KUKA KRL program: f1_Kuka_APT230T02S30.SRC

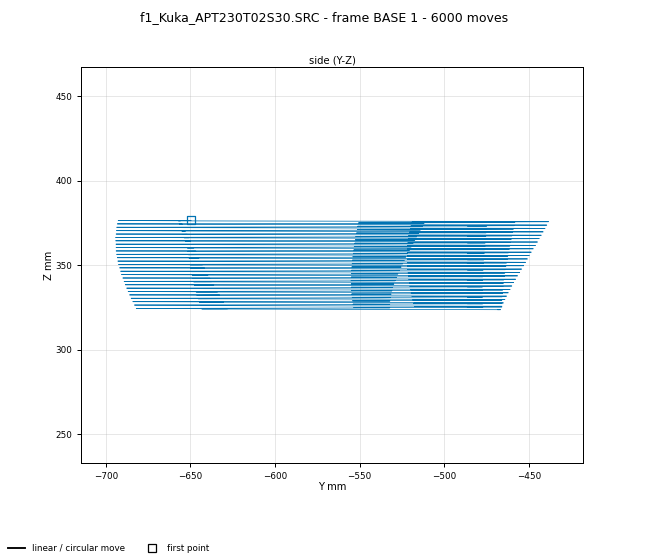
[picture p0: tool path of f1_Kuka_APT230T02S30.SRC in frame BASE 1, 6000 of 6001 moves have a stored position in this frame; points joined in program order, loops and branches not executed]
&ACCESS RVP
&REL 2
&PARAM TEMPLATE = C:\KRC\Roboter\Template\vorgabe
&PARAM EDITMASK = *
DEF f1_Kuka_APT230T02S30()


;FOLD INI;%{PE}%V3.2.0,%MKUKATPBASIS,%CINIT,%VCOMMON,%P
  ;FOLD BAS INI;%{E}%V3.2.0,%MKUKATPBASIS,%CINIT,%VINIT,%P
    GLOBAL INTERRUPT DECL 3 WHEN $STOPMESS==TRUE DO IR_STOPM ( )
    INTERRUPT ON 3
    BAS (#INITMOV,0 )
  ;ENDFOLD (BAS INI)
  ;FOLD USER INI;%{E}%V3.2.0,%MKUKATPUSER,%CINIT,%VINIT,%P
    ;Make your modifications here
  ;ENDFOLD (USER INI)
;ENDFOLD (INI)


;*** Make Null PTP Move
  PTP $pos_act

;*** Auto Load The Correct TOOL Data
  $tool=tool_data[2]

;*** Auto Load The Correct BASE Data
  $base=base_data[1]

  $ADVANCE = 5

;*** Restate Last Velocity
MMPM(30000.0)
SetRPM(8000)
LIN {X 0.163,Y -649.704,Z 376.543,A 0.000,B 0.000,C 90.000,E1 313.704} C_DIS
LIN {X -0.056,Y -653.378,Z 376.537,A 0.000,B 0.000,C 90.000,E1 312.732} C_DIS
LIN {X 0.228,Y -658.806,Z 376.529,A 0.000,B 0.000,C 90.000,E1 311.229} C_DIS
LIN {X 0.152,Y -663.209,Z 376.522,A 0.000,B 0.000,C 90.000,E1 310.011} C_DIS
LIN {X 0.173,Y -665.779,Z 376.518,A 0.000,B 0.000,C 90.000,E1 309.277} C_DIS
LIN {X -0.223,Y -669.831,Z 376.512,A 0.000,B 0.000,C 90.000,E1 308.096} C_DIS
LIN {X -0.019,Y -673.030,Z 376.506,A 0.000,B 0.000,C 90.000,E1 307.111} C_DIS
LIN {X 0.091,Y -676.010,Z 376.501,A 0.000,B 0.000,C 90.000,E1 306.137} C_DIS
LIN {X -0.172,Y -678.143,Z 376.497,A 0.000,B 0.000,C 90.000,E1 305.438} C_DIS
LIN {X 0.146,Y -680.171,Z 376.493,A 0.000,B 0.000,C 90.000,E1 304.692} C_DIS
LIN {X 0.314,Y -681.620,Z 376.490,A 0.000,B 0.000,C 90.000,E1 304.199} C_DIS
LIN {X -0.083,Y -684.557,Z 376.484,A 0.000,B 0.000,C 90.000,E1 303.038} C_DIS
LIN {X 0.141,Y -687.938,Z 376.476,A 0.000,B 0.000,C 90.000,E1 301.592} C_DIS
LIN {X 0.208,Y -689.459,Z 376.472,A 0.000,B 0.000,C 90.000,E1 300.875} C_DIS
LIN {X -0.299,Y -690.732,Z 376.468,A 0.000,B 0.000,C 90.000,E1 300.207} C_DIS
LIN {X 0.146,Y -691.673,Z 376.464,A 0.000,B 0.000,C 90.000,E1 299.461} C_DIS
LIN {X 0.255,Y -692.307,Z 376.460,A 0.000,B 0.000,C 90.000,E1 298.743} C_DIS
LIN {X 0.046,Y -692.607,Z 376.456,A 0.000,B 0.000,C 90.000,E1 298.052} C_DIS
LIN {X -0.076,Y -692.747,Z 376.453,A 0.000,B 0.000,C 90.000,E1 297.590} C_DIS
LIN {X 0.045,Y -692.691,Z 376.449,A 0.000,B 0.000,C 90.000,E1 296.873} C_DIS
LIN {X 0.291,Y -692.484,Z 376.448,A 0.000,B 0.000,C 90.000,E1 296.616} C_DIS
LIN {X 0.159,Y -692.369,Z 376.445,A 0.000,B 0.000,C 90.000,E1 296.155} C_DIS
LIN {X 0.154,Y -691.580,Z 376.439,A 0.000,B 0.000,C 90.000,E1 294.975} C_DIS
LIN {X 0.199,Y -690.341,Z 376.434,A 0.000,B 0.000,C 90.000,E1 294.027} C_DIS
LIN {X 0.179,Y -688.376,Z 376.427,A 0.000,B 0.000,C 90.000,E1 292.845} C_DIS
LIN {X 0.168,Y -686.612,Z 376.422,A 0.000,B 0.000,C 90.000,E1 291.897} C_DIS
LIN {X 0.028,Y -683.516,Z 376.414,A 0.000,B 0.000,C 90.000,E1 290.482} C_DIS
LIN {X 0.281,Y -680.993,Z 376.407,A 0.000,B 0.000,C 90.000,E1 289.268} C_DIS
LIN {X -0.153,Y -678.267,Z 376.401,A 0.000,B 0.000,C 90.000,E1 288.109} C_DIS
LIN {X -0.199,Y -675.630,Z 376.394,A 0.000,B 0.000,C 90.000,E1 286.913} C_DIS
LIN {X 0.305,Y -672.527,Z 376.386,A 0.000,B 0.000,C 90.000,E1 285.426} C_DIS
LIN {X 0.074,Y -666.335,Z 376.368,A 0.000,B 0.000,C 90.000,E1 282.299} C_DIS
LIN {X -0.156,Y -661.494,Z 376.351,A 0.000,B 0.000,C 90.000,E1 279.151} C_DIS
LIN {X 0.314,Y -657.922,Z 376.332,A 0.000,B 0.000,C 90.000,E1 275.682} C_DIS
LIN {X -0.180,Y -656.502,Z 376.318,A 0.000,B 0.000,C 90.000,E1 273.269} C_DIS
LIN {X -0.289,Y -655.863,Z 376.303,A 0.000,B 0.000,C 90.000,E1 270.573} C_DIS
LIN {X -0.067,Y -655.914,Z 376.291,A 0.000,B 0.000,C 90.000,E1 268.339} C_DIS
LIN {X 0.196,Y -656.501,Z 376.279,A 0.000,B 0.000,C 90.000,E1 266.102} C_DIS
LIN {X 0.156,Y -656.858,Z 376.273,A 0.000,B 0.000,C 90.000,E1 265.122} C_DIS
LIN {X 0.066,Y -657.098,Z 376.268,A 0.000,B 0.000,C 90.000,E1 264.147} C_DIS
LIN {X -0.089,Y -657.122,Z 376.261,A 0.000,B 0.000,C 90.000,E1 262.932} C_DIS
LIN {X 0.014,Y -656.948,Z 376.257,A 0.000,B 0.000,C 90.000,E1 262.186} C_DIS
LIN {X 0.078,Y -656.478,Z 376.251,A 0.000,B 0.000,C 90.000,E1 261.197} C_DIS
LIN {X -0.265,Y -656.044,Z 376.248,A 0.000,B 0.000,C 90.000,E1 260.735} C_DIS
LIN {X -0.049,Y -653.895,Z 376.239,A 0.000,B 0.000,C 90.000,E1 258.993} C_DIS
LIN {X -0.171,Y -653.502,Z 376.238,A 0.000,B 0.000,C 90.000,E1 258.757} C_DIS
LIN {X 0.226,Y -653.064,Z 376.235,A 0.000,B 0.000,C 90.000,E1 258.229} C_DIS
LIN {X -0.141,Y -651.961,Z 376.231,A 0.000,B 0.000,C 90.000,E1 257.521} C_DIS
LIN {X 0.248,Y -651.310,Z 376.228,A 0.000,B 0.000,C 90.000,E1 256.992} C_DIS
LIN {X 0.374,Y -649.587,Z 376.222,A 0.000,B 0.000,C 90.000,E1 255.992} C_DIS
LIN {X 0.113,Y -648.593,Z 376.220,A 0.000,B 0.000,C 90.000,E1 255.519} C_DIS
LIN {X 0.195,Y -646.368,Z 376.214,A 0.000,B 0.000,C 90.000,E1 254.519} C_DIS
LIN {X -0.057,Y -644.432,Z 376.210,A 0.000,B 0.000,C 90.000,E1 253.795} C_DIS
LIN {X 0.107,Y -642.226,Z 376.206,A 0.000,B 0.000,C 90.000,E1 253.032} C_DIS
LIN {X -0.149,Y -639.008,Z 376.200,A 0.000,B 0.000,C 90.000,E1 252.054} C_DIS
LIN {X 0.143,Y -636.488,Z 376.196,A 0.000,B 0.000,C 90.000,E1 251.275} C_DIS
LIN {X -0.170,Y -632.779,Z 376.190,A 0.000,B 0.000,C 90.000,E1 250.296} C_DIS
LIN {X -0.147,Y -627.965,Z 376.183,A 0.000,B 0.000,C 90.000,E1 249.028} C_DIS
LIN {X 0.239,Y -623.929,Z 376.178,A 0.000,B 0.000,C 90.000,E1 247.975} C_DIS
LIN {X -0.254,Y -618.652,Z 376.171,A 0.000,B 0.000,C 90.000,E1 246.741} C_DIS
LIN {X 0.226,Y -613.303,Z 376.164,A 0.000,B 0.000,C 90.000,E1 245.409} C_DIS
LIN {X -0.239,Y -606.742,Z 376.155,A 0.000,B 0.000,C 90.000,E1 243.896} C_DIS
LIN {X 0.242,Y -600.208,Z 376.146,A 0.000,B 0.000,C 90.000,E1 242.281} C_DIS
LIN {X -0.034,Y -592.621,Z 376.136,A 0.000,B 0.000,C 90.000,E1 240.461} C_DIS
LIN {X -0.159,Y -583.246,Z 376.123,A 0.000,B 0.000,C 90.000,E1 238.074} C_DIS
LIN {X 0.202,Y -575.502,Z 376.111,A 0.000,B 0.000,C 90.000,E1 235.881} C_DIS
LIN {X -0.064,Y -569.970,Z 376.102,A 0.000,B 0.000,C 90.000,E1 234.276} C_DIS
LIN {X -0.226,Y -565.448,Z 376.094,A 0.000,B 0.000,C 90.000,E1 232.924} C_DIS
LIN {X -0.227,Y -561.722,Z 376.088,A 0.000,B 0.000,C 90.000,E1 231.823} C_DIS
LIN {X -0.109,Y -555.912,Z 376.079,A 0.000,B 0.000,C 90.000,E1 230.150} C_DIS
LIN {X 0.223,Y -549.385,Z 376.068,A 0.000,B 0.000,C 90.000,E1 228.162} C_DIS
LIN {X -0.030,Y -544.865,Z 376.060,A 0.000,B 0.000,C 90.000,E1 226.782} C_DIS
LIN {X 0.002,Y -540.354,Z 376.052,A 0.000,B 0.000,C 90.000,E1 225.364} C_DIS
LIN {X -0.058,Y -534.992,Z 376.043,A 0.000,B 0.000,C 90.000,E1 223.662} C_DIS
LIN {X 0.145,Y -529.675,Z 376.033,A 0.000,B 0.000,C 90.000,E1 221.919} C_DIS
LIN {X -0.215,Y -522.839,Z 376.020,A 0.000,B 0.000,C 90.000,E1 219.644} C_DIS
LIN {X -0.174,Y -517.905,Z 376.010,A 0.000,B 0.000,C 90.000,E1 217.890} C_DIS
LIN {X 0.166,Y -513.141,Z 376.001,A 0.000,B 0.000,C 90.000,E1 216.091} C_DIS
LIN {X -0.003,Y -507.832,Z 375.989,A 0.000,B 0.000,C 90.000,E1 214.040} C_DIS
LIN {X -0.025,Y -502.737,Z 375.978,A 0.000,B 0.000,C 90.000,E1 211.957} C_DIS
LIN {X 0.071,Y -499.981,Z 375.971,A 0.000,B 0.000,C 90.000,E1 210.747} C_DIS
LIN {X 0.005,Y -495.857,Z 375.961,A 0.000,B 0.000,C 90.000,E1 208.949} C_DIS
LIN {X 0.061,Y -491.070,Z 375.949,A 0.000,B 0.000,C 90.000,E1 206.821} C_DIS
LIN {X -0.019,Y -486.141,Z 375.937,A 0.000,B 0.000,C 90.000,E1 204.695} C_DIS
LIN {X 0.039,Y -482.460,Z 375.929,A 0.000,B 0.000,C 90.000,E1 203.153} C_DIS
LIN {X 0.222,Y -478.781,Z 375.920,A 0.000,B 0.000,C 90.000,E1 201.589} C_DIS
LIN {X -0.045,Y -474.447,Z 375.910,A 0.000,B 0.000,C 90.000,E1 199.758} C_DIS
LIN {X -0.204,Y -468.870,Z 375.896,A 0.000,B 0.000,C 90.000,E1 197.275} C_DIS
LIN {X -0.082,Y -464.978,Z 375.885,A 0.000,B 0.000,C 90.000,E1 195.371} C_DIS
LIN {X 0.184,Y -460.689,Z 375.873,A 0.000,B 0.000,C 90.000,E1 193.119} C_DIS
LIN {X 0.121,Y -455.523,Z 375.857,A 0.000,B 0.000,C 90.000,E1 190.254} C_DIS
LIN {X -0.237,Y -451.787,Z 375.845,A 0.000,B 0.000,C 90.000,E1 188.049} C_DIS
LIN {X 0.137,Y -448.336,Z 375.832,A 0.000,B 0.000,C 90.000,E1 185.739} C_DIS
LIN {X -0.039,Y -442.797,Z 375.807,A 0.000,B 0.000,C 90.000,E1 181.203} C_DIS
LIN {X -0.001,Y -439.945,Z 375.787,A 0.000,B 0.000,C 90.000,E1 177.593} C_DIS
LIN {X -0.171,Y -438.299,Z 375.763,A 0.000,B 0.000,C 90.000,E1 173.337} C_DIS
LIN {X -0.004,Y -438.509,Z 375.737,A 0.000,B 0.000,C 90.000,E1 168.701} C_DIS
LIN {X 0.032,Y -442.330,Z 375.704,A 0.000,B 0.000,C 90.000,E1 162.779} C_DIS
LIN {X -0.158,Y -446.351,Z 375.684,A 0.000,B 0.000,C 90.000,E1 159.209} C_DIS
LIN {X 0.123,Y -452.263,Z 375.663,A 0.000,B 0.000,C 90.000,E1 155.281} C_DIS
LIN {X -0.157,Y -455.693,Z 375.652,A 0.000,B 0.000,C 90.000,E1 153.384} C_DIS
LIN {X -0.048,Y -463.942,Z 375.631,A 0.000,B 0.000,C 90.000,E1 149.537} C_DIS
LIN {X -0.201,Y -473.215,Z 375.612,A 0.000,B 0.000,C 90.000,E1 146.087} C_DIS
LIN {X -0.040,Y -481.024,Z 375.598,A 0.000,B 0.000,C 90.000,E1 143.577} C_DIS
LIN {X -0.174,Y -487.223,Z 375.587,A 0.000,B 0.000,C 90.000,E1 141.743} C_DIS
LIN {X -0.003,Y -492.431,Z 375.579,A 0.000,B 0.000,C 90.000,E1 140.194} C_DIS
LIN {X 0.032,Y -496.524,Z 375.572,A 0.000,B 0.000,C 90.000,E1 138.976} C_DIS
LIN {X 0.131,Y -500.477,Z 375.565,A 0.000,B 0.000,C 90.000,E1 137.757} C_DIS
LIN {X -0.085,Y -504.202,Z 375.559,A 0.000,B 0.000,C 90.000,E1 136.581} C_DIS
LIN {X 0.236,Y -506.818,Z 375.554,A 0.000,B 0.000,C 90.000,E1 135.648} C_DIS
LIN {X -0.258,Y -509.980,Z 375.547,A 0.000,B 0.000,C 90.000,E1 134.514} C_DIS
LIN {X 0.233,Y -511.429,Z 375.544,A 0.000,B 0.000,C 90.000,E1 133.866} C_DIS
LIN {X -0.086,Y -513.399,Z 375.539,A 0.000,B 0.000,C 90.000,E1 133.014} C_DIS
LIN {X 0.085,Y -514.607,Z 375.536,A 0.000,B 0.000,C 90.000,E1 132.405} C_DIS
LIN {X 0.145,Y -516.140,Z 375.531,A 0.000,B 0.000,C 90.000,E1 131.515} C_DIS
LIN {X 0.265,Y -517.444,Z 375.526,A 0.000,B 0.000,C 90.000,E1 130.620} C_DIS
LIN {X 0.003,Y -518.419,Z 375.521,A 0.000,B 0.000,C 90.000,E1 129.769} C_DIS
LIN {X 0.085,Y -519.013,Z 375.514,A 0.000,B 0.000,C 90.000,E1 128.588} C_DIS
LIN {X -0.144,Y -518.670,Z 375.508,A 0.000,B 0.000,C 90.000,E1 127.443} C_DIS
LIN {X -0.317,Y -518.081,Z 375.503,A 0.000,B 0.000,C 90.000,E1 126.583} C_DIS
LIN {X -0.016,Y -517.558,Z 375.500,A 0.000,B 0.000,C 90.000,E1 125.964} C_DIS
LIN {X -0.199,Y -516.417,Z 375.495,A 0.000,B 0.000,C 90.000,E1 125.105} C_DIS
LIN {X 0.025,Y -515.035,Z 375.490,A 0.000,B 0.000,C 90.000,E1 124.199} C_DIS
LIN {X 0.230,Y -513.407,Z 375.485,A 0.000,B 0.000,C 90.000,E1 123.293} C_DIS
LIN {X 0.135,Y -511.551,Z 375.480,A 0.000,B 0.000,C 90.000,E1 122.418} C_DIS
LIN {X 0.025,Y -509.351,Z 375.475,A 0.000,B 0.000,C 90.000,E1 121.544} C_DIS
LIN {X 0.215,Y -505.989,Z 375.469,A 0.000,B 0.000,C 90.000,E1 120.335} C_DIS
LIN {X 0.037,Y -503.218,Z 375.464,A 0.000,B 0.000,C 90.000,E1 119.461} C_DIS
LIN {X -0.036,Y -501.245,Z 375.460,A 0.000,B 0.000,C 90.000,E1 118.871} C_DIS
LIN {X -0.070,Y -497.929,Z 375.455,A 0.000,B 0.000,C 90.000,E1 117.975} C_DIS
LIN {X 0.091,Y -494.389,Z 375.450,A 0.000,B 0.000,C 90.000,E1 117.052} C_DIS
LIN {X 0.008,Y -489.325,Z 375.444,A 0.000,B 0.000,C 90.000,E1 115.848} C_DIS
LIN {X -0.162,Y -485.364,Z 375.439,A 0.000,B 0.000,C 90.000,E1 114.951} C_DIS
LIN {X -0.137,Y -481.107,Z 375.433,A 0.000,B 0.000,C 90.000,E1 114.027} C_DIS
LIN {X 0.019,Y -475.347,Z 375.427,A 0.000,B 0.000,C 90.000,E1 112.770} C_DIS
LIN {X 0.096,Y -468.465,Z 375.419,A 0.000,B 0.000,C 90.000,E1 111.354} C_DIS
LIN {X 0.172,Y -458.226,Z 375.407,A 0.000,B 0.000,C 90.000,E1 109.268} C_DIS
LIN {X 0.132,Y -458.213,Z 375.407,A 0.000,B 0.000,C 90.000,E1 109.268} C_DIS
LIN {X -0.112,Y -467.081,Z 375.384,A 0.000,B 0.000,C 90.000,E1 105.190} C_DIS
LIN {X 0.263,Y -467.845,Z 375.383,A 0.000,B 0.000,C 90.000,E1 104.828} C_DIS
LIN {X -0.176,Y -475.403,Z 375.358,A 0.000,B 0.000,C 90.000,E1 100.489} C_DIS
LIN {X 0.130,Y -476.055,Z 375.356,A 0.000,B 0.000,C 90.000,E1 100.141} C_DIS
LIN {X -0.066,Y -481.981,Z 375.331,A 0.000,B 0.000,C 90.000,E1 95.511} C_DIS
LIN {X 0.068,Y -482.357,Z 375.327,A 0.000,B 0.000,C 90.000,E1 94.878} C_DIS
LIN {X 0.205,Y -485.435,Z 375.305,A 0.000,B 0.000,C 90.000,E1 90.859} C_DIS
LIN {X -0.143,Y -485.505,Z 375.302,A 0.000,B 0.000,C 90.000,E1 90.286} C_DIS
LIN {X 0.238,Y -486.377,Z 375.281,A 0.000,B 0.000,C 90.000,E1 86.560} C_DIS
LIN {X 0.062,Y -486.365,Z 375.279,A 0.000,B 0.000,C 90.000,E1 86.274} C_DIS
LIN {X 0.151,Y -484.691,Z 375.254,A 0.000,B 0.000,C 90.000,E1 81.659} C_DIS
LIN {X -0.052,Y -484.454,Z 375.252,A 0.000,B 0.000,C 90.000,E1 81.376} C_DIS
LIN {X -0.048,Y -480.646,Z 375.228,A 0.000,B 0.000,C 90.000,E1 77.061} C_DIS
LIN {X -0.081,Y -480.368,Z 375.226,A 0.000,B 0.000,C 90.000,E1 76.756} C_DIS
LIN {X 0.233,Y -474.654,Z 375.203,A 0.000,B 0.000,C 90.000,E1 72.543} C_DIS
LIN {X 0.192,Y -474.657,Z 375.203,A 0.000,B 0.000,C 90.000,E1 72.543} C_DIS
LIN {X -0.287,Y -485.495,Z 375.195,A 0.000,B 0.000,C 90.000,E1 71.040} C_DIS
LIN {X 0.252,Y -493.631,Z 375.188,A 0.000,B 0.000,C 90.000,E1 69.752} C_DIS
LIN {X -0.242,Y -499.267,Z 375.183,A 0.000,B 0.000,C 90.000,E1 68.901} C_DIS
LIN {X 0.087,Y -501.950,Z 375.180,A 0.000,B 0.000,C 90.000,E1 68.411} C_DIS
LIN {X 0.051,Y -506.035,Z 375.176,A 0.000,B 0.000,C 90.000,E1 67.667} C_DIS
LIN {X 0.236,Y -509.004,Z 375.173,A 0.000,B 0.000,C 90.000,E1 67.050} C_DIS
LIN {X 0.155,Y -511.255,Z 375.170,A 0.000,B 0.000,C 90.000,E1 66.613} C_DIS
LIN {X 0.087,Y -513.235,Z 375.168,A 0.000,B 0.000,C 90.000,E1 66.177} C_DIS
LIN {X -0.091,Y -514.004,Z 375.167,A 0.000,B 0.000,C 90.000,E1 66.049} C_DIS
LIN {X -0.146,Y -515.847,Z 375.164,A 0.000,B 0.000,C 90.000,E1 65.613} C_DIS
LIN {X -0.322,Y -516.567,Z 375.164,A 0.000,B 0.000,C 90.000,E1 65.485} C_DIS
LIN {X -0.179,Y -519.975,Z 375.159,A 0.000,B 0.000,C 90.000,E1 64.588} C_DIS
LIN {X 0.099,Y -522.152,Z 375.156,A 0.000,B 0.000,C 90.000,E1 63.973} C_DIS
LIN {X 0.153,Y -524.176,Z 375.152,A 0.000,B 0.000,C 90.000,E1 63.384} C_DIS
LIN {X -0.085,Y -526.875,Z 375.147,A 0.000,B 0.000,C 90.000,E1 62.538} C_DIS
LIN {X -0.128,Y -530.387,Z 375.141,A 0.000,B 0.000,C 90.000,E1 61.385} C_DIS
LIN {X 0.129,Y -533.596,Z 375.135,A 0.000,B 0.000,C 90.000,E1 60.205} C_DIS
LIN {X -0.039,Y -537.417,Z 375.127,A 0.000,B 0.000,C 90.000,E1 58.791} C_DIS
LIN {X 0.136,Y -539.558,Z 375.122,A 0.000,B 0.000,C 90.000,E1 57.916} C_DIS
LIN {X 0.075,Y -542.930,Z 375.114,A 0.000,B 0.000,C 90.000,E1 56.501} C_DIS
LIN {X -0.118,Y -545.358,Z 375.108,A 0.000,B 0.000,C 90.000,E1 55.388} C_DIS
LIN {X -0.003,Y -546.950,Z 375.103,A 0.000,B 0.000,C 90.000,E1 54.529} C_DIS
LIN {X -0.142,Y -548.586,Z 375.097,A 0.000,B 0.000,C 90.000,E1 53.417} C_DIS
LIN {X 0.064,Y -549.837,Z 375.090,A 0.000,B 0.000,C 90.000,E1 52.271} C_DIS
LIN {X 0.117,Y -550.121,Z 375.089,A 0.000,B 0.000,C 90.000,E1 51.984} C_DIS
LIN {X -0.093,Y -550.614,Z 375.083,A 0.000,B 0.000,C 90.000,E1 50.884} C_DIS
LIN {X 0.000,Y -550.587,Z 375.078,A 0.000,B 0.000,C 90.000,E1 50.033} C_DIS
LIN {X 0.160,Y -550.371,Z 375.073,A 0.000,B 0.000,C 90.000,E1 49.175} C_DIS
LIN {X 0.254,Y -549.766,Z 375.069,A 0.000,B 0.000,C 90.000,E1 48.324} C_DIS
LIN {X -0.020,Y -548.559,Z 375.062,A 0.000,B 0.000,C 90.000,E1 47.229} C_DIS
LIN {X -0.309,Y -546.986,Z 375.056,A 0.000,B 0.000,C 90.000,E1 46.134} C_DIS
LIN {X 0.180,Y -544.249,Z 375.045,A 0.000,B 0.000,C 90.000,E1 44.109} C_DIS
LIN {X -0.167,Y -541.850,Z 375.036,A 0.000,B 0.000,C 90.000,E1 42.447} C_DIS
LIN {X -0.147,Y -538.823,Z 375.023,A 0.000,B 0.000,C 90.000,E1 40.172} C_DIS
LIN {X -0.156,Y -536.567,Z 375.014,A 0.000,B 0.000,C 90.000,E1 38.463} C_DIS
LIN {X -0.122,Y -534.379,Z 375.004,A 0.000,B 0.000,C 90.000,E1 36.744} C_DIS
LIN {X -0.131,Y -532.446,Z 374.996,A 0.000,B 0.000,C 90.000,E1 35.311} C_DIS
LIN {X -0.065,Y -530.203,Z 374.987,A 0.000,B 0.000,C 90.000,E1 33.579} C_DIS
LIN {X 0.079,Y -527.648,Z 374.975,A 0.000,B 0.000,C 90.000,E1 31.544} C_DIS
LIN {X 0.193,Y -525.508,Z 374.966,A 0.000,B 0.000,C 90.000,E1 29.795} C_DIS
LIN {X 0.052,Y -523.803,Z 374.958,A 0.000,B 0.000,C 90.000,E1 28.359} C_DIS
LIN {X -0.123,Y -522.169,Z 374.950,A 0.000,B 0.000,C 90.000,E1 26.924} C_DIS
LIN {X 0.048,Y -520.324,Z 374.940,A 0.000,B 0.000,C 90.000,E1 25.155} C_DIS
LIN {X -0.154,Y -518.289,Z 374.928,A 0.000,B 0.000,C 90.000,E1 23.131} C_DIS
LIN {X 0.059,Y -515.807,Z 374.912,A 0.000,B 0.000,C 90.000,E1 20.174} C_DIS
LIN {X 0.189,Y -514.050,Z 374.897,A 0.000,B 0.000,C 90.000,E1 17.511} C_DIS
LIN {X -0.178,Y -512.754,Z 374.883,A 0.000,B 0.000,C 90.000,E1 14.898} C_DIS
LIN {X -0.175,Y -512.069,Z 374.870,A 0.000,B 0.000,C 90.000,E1 12.535} C_DIS
LIN {X -0.004,Y -511.885,Z 374.852,A 0.000,B 0.000,C 90.000,E1 9.265} C_DIS
LIN {X 0.081,Y -512.308,Z 374.838,A 0.000,B 0.000,C 90.000,E1 6.891} C_DIS
LIN {X -0.024,Y -513.453,Z 374.824,A 0.000,B 0.000,C 90.000,E1 4.245} C_DIS
LIN {X -0.127,Y -515.362,Z 374.809,A 0.000,B 0.000,C 90.000,E1 1.604} C_DIS
LIN {X 0.244,Y -520.032,Z 374.786,A 0.000,B 0.000,C 90.000,E1 357.421} C_DIS
LIN {X -0.073,Y -523.075,Z 374.775,A 0.000,B 0.000,C 90.000,E1 355.412} C_DIS
LIN {X -0.271,Y -527.127,Z 374.762,A 0.000,B 0.000,C 90.000,E1 353.109} C_DIS
LIN {X -0.090,Y -534.841,Z 374.741,A 0.000,B 0.000,C 90.000,E1 349.342} C_DIS
LIN {X -0.169,Y -544.480,Z 374.720,A 0.000,B 0.000,C 90.000,E1 345.644} C_DIS
LIN {X 0.116,Y -549.305,Z 374.711,A 0.000,B 0.000,C 90.000,E1 343.921} C_DIS
LIN {X -0.129,Y -553.486,Z 374.703,A 0.000,B 0.000,C 90.000,E1 342.543} C_DIS
LIN {X -0.018,Y -558.490,Z 374.694,A 0.000,B 0.000,C 90.000,E1 340.859} C_DIS
LIN {X -0.145,Y -563.565,Z 374.684,A 0.000,B 0.000,C 90.000,E1 339.209} C_DIS
LIN {X -0.103,Y -566.884,Z 374.678,A 0.000,B 0.000,C 90.000,E1 338.103} C_DIS
LIN {X -0.196,Y -571.087,Z 374.671,A 0.000,B 0.000,C 90.000,E1 336.741} C_DIS
LIN {X 0.221,Y -576.931,Z 374.660,A 0.000,B 0.000,C 90.000,E1 334.793} C_DIS
LIN {X 0.256,Y -584.689,Z 374.647,A 0.000,B 0.000,C 90.000,E1 332.359} C_DIS
LIN {X -0.008,Y -590.966,Z 374.636,A 0.000,B 0.000,C 90.000,E1 330.511} C_DIS
LIN {X -0.023,Y -596.400,Z 374.627,A 0.000,B 0.000,C 90.000,E1 328.918} C_DIS
LIN {X 0.150,Y -600.909,Z 374.620,A 0.000,B 0.000,C 90.000,E1 327.582} C_DIS
LIN {X -0.249,Y -609.062,Z 374.607,A 0.000,B 0.000,C 90.000,E1 325.261} C_DIS
LIN {X -0.255,Y -614.717,Z 374.598,A 0.000,B 0.000,C 90.000,E1 323.703} C_DIS
LIN {X -0.086,Y -619.511,Z 374.591,A 0.000,B 0.000,C 90.000,E1 322.396} C_DIS
LIN {X -0.038,Y -626.267,Z 374.581,A 0.000,B 0.000,C 90.000,E1 320.598} C_DIS
LIN {X -0.053,Y -633.951,Z 374.570,A 0.000,B 0.000,C 90.000,E1 318.566} C_DIS
LIN {X -0.010,Y -637.576,Z 374.564,A 0.000,B 0.000,C 90.000,E1 317.553} C_DIS
LIN {X -0.001,Y -642.053,Z 374.557,A 0.000,B 0.000,C 90.000,E1 316.296} C_DIS
LIN {X 0.009,Y -647.512,Z 374.549,A 0.000,B 0.000,C 90.000,E1 314.798} C_DIS
LIN {X 0.232,Y -651.255,Z 374.543,A 0.000,B 0.000,C 90.000,E1 313.785} C_DIS
LIN {X 0.035,Y -654.898,Z 374.538,A 0.000,B 0.000,C 90.000,E1 312.813} C_DIS
LIN {X -0.145,Y -660.269,Z 374.530,A 0.000,B 0.000,C 90.000,E1 311.353} C_DIS
LIN {X 0.301,Y -664.678,Z 374.523,A 0.000,B 0.000,C 90.000,E1 310.092} C_DIS
LIN {X 0.324,Y -667.978,Z 374.518,A 0.000,B 0.000,C 90.000,E1 309.116} C_DIS
LIN {X -0.033,Y -671.294,Z 374.512,A 0.000,B 0.000,C 90.000,E1 308.177} C_DIS
LIN {X -0.346,Y -674.428,Z 374.507,A 0.000,B 0.000,C 90.000,E1 307.237} C_DIS
LIN {X -0.218,Y -676.731,Z 374.503,A 0.000,B 0.000,C 90.000,E1 306.503} C_DIS
LIN {X -0.075,Y -678.075,Z 374.500,A 0.000,B 0.000,C 90.000,E1 306.011} C_DIS
LIN {X 0.076,Y -678.886,Z 374.499,A 0.000,B 0.000,C 90.000,E1 305.758} C_DIS
LIN {X -0.316,Y -680.131,Z 374.496,A 0.000,B 0.000,C 90.000,E1 305.311} C_DIS
LIN {X 0.241,Y -680.923,Z 374.495,A 0.000,B 0.000,C 90.000,E1 305.025} C_DIS
LIN {X 0.026,Y -682.130,Z 374.492,A 0.000,B 0.000,C 90.000,E1 304.565} C_DIS
LIN {X 0.027,Y -682.928,Z 374.491,A 0.000,B 0.000,C 90.000,E1 304.326} C_DIS
LIN {X -0.171,Y -683.973,Z 374.488,A 0.000,B 0.000,C 90.000,E1 303.865} C_DIS
LIN {X -0.172,Y -684.619,Z 374.487,A 0.000,B 0.000,C 90.000,E1 303.627} C_DIS
LIN {X 0.048,Y -687.207,Z 374.480,A 0.000,B 0.000,C 90.000,E1 302.418} C_DIS
LIN {X -0.118,Y -688.810,Z 374.476,A 0.000,B 0.000,C 90.000,E1 301.720} C_DIS
LIN {X -0.045,Y -690.254,Z 374.472,A 0.000,B 0.000,C 90.000,E1 301.003} C_DIS
LIN {X 0.051,Y -691.474,Z 374.468,A 0.000,B 0.000,C 90.000,E1 300.285} C_DIS
LIN {X -0.095,Y -692.431,Z 374.464,A 0.000,B 0.000,C 90.000,E1 299.589} C_DIS
LIN {X 0.020,Y -693.067,Z 374.460,A 0.000,B 0.000,C 90.000,E1 298.871} C_DIS
LIN {X 0.143,Y -693.216,Z 374.457,A 0.000,B 0.000,C 90.000,E1 298.153} C_DIS
LIN {X -0.301,Y -693.231,Z 374.454,A 0.000,B 0.000,C 90.000,E1 297.719} C_DIS
LIN {X -0.176,Y -692.973,Z 374.450,A 0.000,B 0.000,C 90.000,E1 297.001} C_DIS
LIN {X -0.058,Y -692.446,Z 374.446,A 0.000,B 0.000,C 90.000,E1 296.283} C_DIS
LIN {X -0.118,Y -692.162,Z 374.445,A 0.000,B 0.000,C 90.000,E1 296.052} C_DIS
LIN {X -0.253,Y -691.801,Z 374.442,A 0.000,B 0.000,C 90.000,E1 295.591} C_DIS
LIN {X 0.229,Y -691.408,Z 374.439,A 0.000,B 0.000,C 90.000,E1 295.079} C_DIS
LIN {X -0.020,Y -690.031,Z 374.434,A 0.000,B 0.000,C 90.000,E1 294.155} C_DIS
LIN {X -0.229,Y -688.898,Z 374.430,A 0.000,B 0.000,C 90.000,E1 293.462} C_DIS
LIN {X -0.272,Y -686.736,Z 374.424,A 0.000,B 0.000,C 90.000,E1 292.280} C_DIS
LIN {X 0.117,Y -685.198,Z 374.420,A 0.000,B 0.000,C 90.000,E1 291.535} C_DIS
LIN {X -0.090,Y -681.444,Z 374.410,A 0.000,B 0.000,C 90.000,E1 289.885} C_DIS
LIN {X 0.139,Y -678.746,Z 374.404,A 0.000,B 0.000,C 90.000,E1 288.671} C_DIS
LIN {X 0.350,Y -674.381,Z 374.393,A 0.000,B 0.000,C 90.000,E1 286.732} C_DIS
LIN {X 0.000,Y -671.261,Z 374.385,A 0.000,B 0.000,C 90.000,E1 285.315} C_DIS
LIN {X 0.041,Y -665.944,Z 374.370,A 0.000,B 0.000,C 90.000,E1 282.647} C_DIS
LIN {X 0.045,Y -663.461,Z 374.362,A 0.000,B 0.000,C 90.000,E1 281.186} C_DIS
LIN {X -0.093,Y -659.689,Z 374.347,A 0.000,B 0.000,C 90.000,E1 278.511} C_DIS
LIN {X 0.214,Y -656.480,Z 374.328,A 0.000,B 0.000,C 90.000,E1 275.049} C_DIS
LIN {X 0.068,Y -655.462,Z 374.317,A 0.000,B 0.000,C 90.000,E1 273.094} C_DIS
LIN {X 0.084,Y -654.906,Z 374.304,A 0.000,B 0.000,C 90.000,E1 270.630} C_DIS
LIN {X -0.094,Y -655.015,Z 374.289,A 0.000,B 0.000,C 90.000,E1 267.936} C_DIS
LIN {X 0.160,Y -655.829,Z 374.276,A 0.000,B 0.000,C 90.000,E1 265.698} C_DIS
LIN {X -0.288,Y -656.363,Z 374.268,A 0.000,B 0.000,C 90.000,E1 264.261} C_DIS
LIN {X 0.121,Y -656.576,Z 374.261,A 0.000,B 0.000,C 90.000,E1 262.996} C_DIS
LIN {X 0.299,Y -656.431,Z 374.257,A 0.000,B 0.000,C 90.000,E1 262.243} C_DIS
LIN {X 0.358,Y -656.092,Z 374.252,A 0.000,B 0.000,C 90.000,E1 261.254} C_DIS
LIN {X 0.012,Y -655.755,Z 374.249,A 0.000,B 0.000,C 90.000,E1 260.792} C_DIS
LIN {X 0.228,Y -654.020,Z 374.239,A 0.000,B 0.000,C 90.000,E1 259.050} C_DIS
LIN {X 0.106,Y -653.691,Z 374.238,A 0.000,B 0.000,C 90.000,E1 258.814} C_DIS
LIN {X -0.256,Y -653.135,Z 374.234,A 0.000,B 0.000,C 90.000,E1 258.105} C_DIS
LIN {X -0.245,Y -651.899,Z 374.228,A 0.000,B 0.000,C 90.000,E1 257.117} C_DIS
LIN {X -0.115,Y -650.436,Z 374.223,A 0.000,B 0.000,C 90.000,E1 256.117} C_DIS
LIN {X -0.372,Y -649.548,Z 374.220,A 0.000,B 0.000,C 90.000,E1 255.644} C_DIS
LIN {X -0.247,Y -646.850,Z 374.213,A 0.000,B 0.000,C 90.000,E1 254.393} C_DIS
LIN {X 0.129,Y -644.939,Z 374.209,A 0.000,B 0.000,C 90.000,E1 253.614} C_DIS
LIN {X -0.316,Y -642.798,Z 374.205,A 0.000,B 0.000,C 90.000,E1 252.906} C_DIS
LIN {X -0.117,Y -638.876,Z 374.198,A 0.000,B 0.000,C 90.000,E1 251.638} C_DIS
LIN {X 0.199,Y -635.393,Z 374.192,A 0.000,B 0.000,C 90.000,E1 250.604} C_DIS
LIN {X -0.326,Y -630.640,Z 374.185,A 0.000,B 0.000,C 90.000,E1 249.390} C_DIS
LIN {X -0.121,Y -625.693,Z 374.178,A 0.000,B 0.000,C 90.000,E1 248.103} C_DIS
LIN {X 0.233,Y -621.553,Z 374.173,A 0.000,B 0.000,C 90.000,E1 247.050} C_DIS
LIN {X -0.071,Y -615.151,Z 374.164,A 0.000,B 0.000,C 90.000,E1 245.537} C_DIS
LIN {X 0.051,Y -608.607,Z 374.155,A 0.000,B 0.000,C 90.000,E1 243.973} C_DIS
LIN {X -0.035,Y -601.037,Z 374.145,A 0.000,B 0.000,C 90.000,E1 242.153} C_DIS
LIN {X -0.200,Y -594.551,Z 374.137,A 0.000,B 0.000,C 90.000,E1 240.589} C_DIS
LIN {X -0.135,Y -586.183,Z 374.125,A 0.000,B 0.000,C 90.000,E1 238.456} C_DIS
LIN {X -0.004,Y -576.438,Z 374.110,A 0.000,B 0.000,C 90.000,E1 235.754} C_DIS
LIN {X 0.081,Y -570.951,Z 374.101,A 0.000,B 0.000,C 90.000,E1 234.116} C_DIS
LIN {X -0.060,Y -566.435,Z 374.093,A 0.000,B 0.000,C 90.000,E1 232.763} C_DIS
LIN {X 0.062,Y -561.712,Z 374.086,A 0.000,B 0.000,C 90.000,E1 231.376} C_DIS
LIN {X -0.172,Y -554.989,Z 374.075,A 0.000,B 0.000,C 90.000,E1 229.461} C_DIS
LIN {X 0.142,Y -548.548,Z 374.064,A 0.000,B 0.000,C 90.000,E1 227.472} C_DIS
LIN {X -0.130,Y -543.153,Z 374.054,A 0.000,B 0.000,C 90.000,E1 225.810} C_DIS
LIN {X 0.232,Y -536.852,Z 374.043,A 0.000,B 0.000,C 90.000,E1 223.785} C_DIS
LIN {X 0.108,Y -531.547,Z 374.034,A 0.000,B 0.000,C 90.000,E1 222.081} C_DIS
LIN {X -0.196,Y -524.653,Z 374.021,A 0.000,B 0.000,C 90.000,E1 219.806} C_DIS
LIN {X 0.210,Y -519.673,Z 374.011,A 0.000,B 0.000,C 90.000,E1 218.016} C_DIS
LIN {X -0.140,Y -514.893,Z 374.002,A 0.000,B 0.000,C 90.000,E1 216.297} C_DIS
LIN {X 0.158,Y -509.521,Z 373.990,A 0.000,B 0.000,C 90.000,E1 214.199} C_DIS
LIN {X 0.029,Y -504.428,Z 373.979,A 0.000,B 0.000,C 90.000,E1 212.133} C_DIS
LIN {X -0.243,Y -500.954,Z 373.970,A 0.000,B 0.000,C 90.000,E1 210.669} C_DIS
LIN {X 0.144,Y -496.849,Z 373.960,A 0.000,B 0.000,C 90.000,E1 208.821} C_DIS
LIN {X -0.213,Y -492.081,Z 373.948,A 0.000,B 0.000,C 90.000,E1 206.744} C_DIS
LIN {X -0.055,Y -487.886,Z 373.938,A 0.000,B 0.000,C 90.000,E1 204.899} C_DIS
LIN {X 0.222,Y -485.008,Z 373.932,A 0.000,B 0.000,C 90.000,E1 203.643} C_DIS
LIN {X -0.177,Y -480.631,Z 373.921,A 0.000,B 0.000,C 90.000,E1 201.844} C_DIS
LIN {X 0.196,Y -475.538,Z 373.909,A 0.000,B 0.000,C 90.000,E1 199.631} C_DIS
LIN {X 0.060,Y -470.016,Z 373.895,A 0.000,B 0.000,C 90.000,E1 197.149} C_DIS
LIN {X 0.007,Y -465.496,Z 373.883,A 0.000,B 0.000,C 90.000,E1 194.954} C_DIS
LIN {X -0.067,Y -461.806,Z 373.873,A 0.000,B 0.000,C 90.000,E1 193.063} C_DIS
LIN {X 0.137,Y -457.217,Z 373.858,A 0.000,B 0.000,C 90.000,E1 190.489} C_DIS
LIN {X 0.130,Y -453.964,Z 373.848,A 0.000,B 0.000,C 90.000,E1 188.568} C_DIS
LIN {X -0.144,Y -449.934,Z 373.833,A 0.000,B 0.000,C 90.000,E1 186.024} C_DIS
LIN {X 0.083,Y -446.794,Z 373.821,A 0.000,B 0.000,C 90.000,E1 183.726} C_DIS
LIN {X 0.024,Y -443.593,Z 373.805,A 0.000,B 0.000,C 90.000,E1 180.802} C_DIS
LIN {X -0.023,Y -441.089,Z 373.786,A 0.000,B 0.000,C 90.000,E1 177.535} C_DIS
LIN {X 0.151,Y -439.443,Z 373.764,A 0.000,B 0.000,C 90.000,E1 173.571} C_DIS
LIN {X -0.077,Y -439.343,Z 373.744,A 0.000,B 0.000,C 90.000,E1 169.982} C_DIS
LIN {X -0.007,Y -440.991,Z 373.721,A 0.000,B 0.000,C 90.000,E1 165.700} C_DIS
LIN {X 0.189,Y -443.418,Z 373.704,A 0.000,B 0.000,C 90.000,E1 162.725} C_DIS
LIN {X -0.247,Y -447.019,Z 373.686,A 0.000,B 0.000,C 90.000,E1 159.518} C_DIS
LIN {X 0.163,Y -450.679,Z 373.672,A 0.000,B 0.000,C 90.000,E1 156.869} C_DIS
LIN {X -0.271,Y -454.378,Z 373.659,A 0.000,B 0.000,C 90.000,E1 154.665} C_DIS
LIN {X -0.172,Y -461.380,Z 373.640,A 0.000,B 0.000,C 90.000,E1 151.129} C_DIS
LIN {X -0.136,Y -470.779,Z 373.618,A 0.000,B 0.000,C 90.000,E1 147.327} C_DIS
LIN {X -0.257,Y -481.138,Z 373.599,A 0.000,B 0.000,C 90.000,E1 143.909} C_DIS
LIN {X 0.002,Y -487.372,Z 373.589,A 0.000,B 0.000,C 90.000,E1 142.029} C_DIS
LIN {X 0.024,Y -493.602,Z 373.579,A 0.000,B 0.000,C 90.000,E1 140.194} C_DIS
LIN {X -0.065,Y -498.628,Z 373.570,A 0.000,B 0.000,C 90.000,E1 138.690} C_DIS
LIN {X -0.144,Y -501.554,Z 373.565,A 0.000,B 0.000,C 90.000,E1 137.796} C_DIS
LIN {X -0.007,Y -505.257,Z 373.559,A 0.000,B 0.000,C 90.000,E1 136.581} C_DIS
LIN {X -0.028,Y -507.827,Z 373.554,A 0.000,B 0.000,C 90.000,E1 135.688} C_DIS
LIN {X -0.153,Y -510.969,Z 373.547,A 0.000,B 0.000,C 90.000,E1 134.514} C_DIS
LIN {X -0.124,Y -513.067,Z 373.542,A 0.000,B 0.000,C 90.000,E1 133.623} C_DIS
LIN {X 0.301,Y -514.910,Z 373.537,A 0.000,B 0.000,C 90.000,E1 132.690} C_DIS
LIN {X 0.020,Y -516.498,Z 373.533,A 0.000,B 0.000,C 90.000,E1 131.838} C_DIS
LIN {X -0.247,Y -517.815,Z 373.528,A 0.000,B 0.000,C 90.000,E1 130.987} C_DIS
LIN {X -0.170,Y -519.089,Z 373.521,A 0.000,B 0.000,C 90.000,E1 129.806} C_DIS
LIN {X -0.070,Y -519.626,Z 373.515,A 0.000,B 0.000,C 90.000,E1 128.624} C_DIS
LIN {X 0.088,Y -519.422,Z 373.510,A 0.000,B 0.000,C 90.000,E1 127.729} C_DIS
LIN {X -0.077,Y -518.913,Z 373.505,A 0.000,B 0.000,C 90.000,E1 126.870} C_DIS
LIN {X -0.247,Y -518.131,Z 373.500,A 0.000,B 0.000,C 90.000,E1 126.011} C_DIS
LIN {X -0.005,Y -516.986,Z 373.495,A 0.000,B 0.000,C 90.000,E1 125.105} C_DIS
LIN {X 0.225,Y -515.618,Z 373.490,A 0.000,B 0.000,C 90.000,E1 124.199} C_DIS
LIN {X -0.276,Y -514.004,Z 373.485,A 0.000,B 0.000,C 90.000,E1 123.372} C_DIS
LIN {X -0.085,Y -512.200,Z 373.480,A 0.000,B 0.000,C 90.000,E1 122.467} C_DIS
LIN {X -0.192,Y -510.042,Z 373.475,A 0.000,B 0.000,C 90.000,E1 121.592} C_DIS
LIN {X 0.073,Y -505.835,Z 373.467,A 0.000,B 0.000,C 90.000,E1 120.079} C_DIS
LIN {X -0.104,Y -502.985,Z 373.462,A 0.000,B 0.000,C 90.000,E1 119.205} C_DIS
LIN {X 0.119,Y -499.881,Z 373.457,A 0.000,B 0.000,C 90.000,E1 118.281} C_DIS
LIN {X 0.070,Y -496.487,Z 373.452,A 0.000,B 0.000,C 90.000,E1 117.385} C_DIS
LIN {X 0.188,Y -493.523,Z 373.448,A 0.000,B 0.000,C 90.000,E1 116.616} C_DIS
LIN {X -0.138,Y -489.215,Z 373.442,A 0.000,B 0.000,C 90.000,E1 115.591} C_DIS
LIN {X 0.133,Y -485.244,Z 373.437,A 0.000,B 0.000,C 90.000,E1 114.643} C_DIS
LIN {X 0.154,Y -482.488,Z 373.434,A 0.000,B 0.000,C 90.000,E1 114.027} C_DIS
LIN {X -0.110,Y -476.886,Z 373.427,A 0.000,B 0.000,C 90.000,E1 112.823} C_DIS
LIN {X -0.009,Y -470.150,Z 373.419,A 0.000,B 0.000,C 90.000,E1 111.408} C_DIS
LIN {X 0.160,Y -462.398,Z 373.410,A 0.000,B 0.000,C 90.000,E1 109.812} C_DIS
LIN {X 0.154,Y -458.661,Z 373.406,A 0.000,B 0.000,C 90.000,E1 109.033} C_DIS
LIN {X 0.114,Y -458.653,Z 373.406,A 0.000,B 0.000,C 90.000,E1 109.033} C_DIS
LIN {X 0.068,Y -467.753,Z 373.383,A 0.000,B 0.000,C 90.000,E1 104.898} C_DIS
LIN {X 0.040,Y -475.959,Z 373.357,A 0.000,B 0.000,C 90.000,E1 100.197} C_DIS
LIN {X 0.190,Y -476.675,Z 373.353,A 0.000,B 0.000,C 90.000,E1 99.557} C_DIS
LIN {X -0.165,Y -481.909,Z 373.331,A 0.000,B 0.000,C 90.000,E1 95.568} C_DIS
LIN {X 0.162,Y -482.201,Z 373.329,A 0.000,B 0.000,C 90.000,E1 95.220} C_DIS
LIN {X 0.101,Y -485.387,Z 373.305,A 0.000,B 0.000,C 90.000,E1 90.917} C_DIS
LIN {X -0.075,Y -485.530,Z 373.303,A 0.000,B 0.000,C 90.000,E1 90.630} C_DIS
LIN {X 0.133,Y -486.356,Z 373.281,A 0.000,B 0.000,C 90.000,E1 86.617} C_DIS
LIN {X -0.042,Y -486.369,Z 373.280,A 0.000,B 0.000,C 90.000,E1 86.331} C_DIS
LIN {X -0.052,Y -485.860,Z 373.275,A 0.000,B 0.000,C 90.000,E1 85.412} C_DIS
LIN {X -0.019,Y -484.692,Z 373.254,A 0.000,B 0.000,C 90.000,E1 81.724} C_DIS
LIN {X -0.150,Y -484.509,Z 373.252,A 0.000,B 0.000,C 90.000,E1 81.432} C_DIS
LIN {X -0.280,Y -480.443,Z 373.227,A 0.000,B 0.000,C 90.000,E1 76.825} C_DIS
LIN {X 0.199,Y -474.841,Z 373.204,A 0.000,B 0.000,C 90.000,E1 72.725} C_DIS
LIN {X 0.158,Y -474.838,Z 373.204,A 0.000,B 0.000,C 90.000,E1 72.725} C_DIS
LIN {X 0.116,Y -484.284,Z 373.197,A 0.000,B 0.000,C 90.000,E1 71.348} C_DIS
LIN {X 0.147,Y -490.307,Z 373.191,A 0.000,B 0.000,C 90.000,E1 70.423} C_DIS
LIN {X -0.126,Y -497.066,Z 373.185,A 0.000,B 0.000,C 90.000,E1 69.390} C_DIS
LIN {X -0.172,Y -501.524,Z 373.181,A 0.000,B 0.000,C 90.000,E1 68.646} C_DIS
LIN {X 0.066,Y -506.326,Z 373.176,A 0.000,B 0.000,C 90.000,E1 67.720} C_DIS
LIN {X 0.256,Y -509.306,Z 373.173,A 0.000,B 0.000,C 90.000,E1 67.102} C_DIS
LIN {X -0.001,Y -512.066,Z 373.170,A 0.000,B 0.000,C 90.000,E1 66.538} C_DIS
LIN {X 0.056,Y -515.207,Z 373.166,A 0.000,B 0.000,C 90.000,E1 65.793} C_DIS
LIN {X -0.164,Y -517.551,Z 373.162,A 0.000,B 0.000,C 90.000,E1 65.229} C_DIS
LIN {X 0.097,Y -519.699,Z 373.159,A 0.000,B 0.000,C 90.000,E1 64.613} C_DIS
LIN {X 0.129,Y -521.756,Z 373.156,A 0.000,B 0.000,C 90.000,E1 64.024} C_DIS
LIN {X -0.137,Y -524.597,Z 373.151,A 0.000,B 0.000,C 90.000,E1 63.179} C_DIS
LIN {X -0.209,Y -528.014,Z 373.145,A 0.000,B 0.000,C 90.000,E1 62.025} C_DIS
LIN {X 0.059,Y -530.564,Z 373.140,A 0.000,B 0.000,C 90.000,E1 61.129} C_DIS
LIN {X -0.144,Y -533.746,Z 373.133,A 0.000,B 0.000,C 90.000,E1 59.999} C_DIS
LIN {X 0.150,Y -537.575,Z 373.125,A 0.000,B 0.000,C 90.000,E1 58.535} C_DIS
LIN {X 0.043,Y -540.420,Z 373.119,A 0.000,B 0.000,C 90.000,E1 57.406} C_DIS
LIN {X -0.192,Y -543.125,Z 373.113,A 0.000,B 0.000,C 90.000,E1 56.294} C_DIS
LIN {X -0.106,Y -545.012,Z 373.108,A 0.000,B 0.000,C 90.000,E1 55.435} C_DIS
LIN {X 0.178,Y -547.198,Z 373.102,A 0.000,B 0.000,C 90.000,E1 54.276} C_DIS
LIN {X 0.314,Y -548.544,Z 373.097,A 0.000,B 0.000,C 90.000,E1 53.417} C_DIS
LIN {X 0.085,Y -549.920,Z 373.091,A 0.000,B 0.000,C 90.000,E1 52.316} C_DIS
LIN {X 0.197,Y -550.524,Z 373.088,A 0.000,B 0.000,C 90.000,E1 51.743} C_DIS
LIN {X -0.060,Y -551.026,Z 373.083,A 0.000,B 0.000,C 90.000,E1 50.928} C_DIS
LIN {X 0.111,Y -551.088,Z 373.078,A 0.000,B 0.000,C 90.000,E1 50.070} C_DIS
LIN {X 0.213,Y -550.925,Z 373.074,A 0.000,B 0.000,C 90.000,E1 49.218} C_DIS
LIN {X 0.000,Y -550.205,Z 373.067,A 0.000,B 0.000,C 90.000,E1 48.119} C_DIS
LIN {X -0.311,Y -549.413,Z 373.063,A 0.000,B 0.000,C 90.000,E1 47.310} C_DIS
LIN {X -0.225,Y -548.366,Z 373.058,A 0.000,B 0.000,C 90.000,E1 46.458} C_DIS
LIN {X -0.073,Y -545.243,Z 373.046,A 0.000,B 0.000,C 90.000,E1 44.190} C_DIS
LIN {X 0.002,Y -542.890,Z 373.036,A 0.000,B 0.000,C 90.000,E1 42.486} C_DIS
LIN {X 0.004,Y -539.841,Z 373.023,A 0.000,B 0.000,C 90.000,E1 40.216} C_DIS
LIN {X 0.006,Y -537.570,Z 373.014,A 0.000,B 0.000,C 90.000,E1 38.508} C_DIS
LIN {X 0.046,Y -535.727,Z 373.006,A 0.000,B 0.000,C 90.000,E1 37.076} C_DIS
LIN {X 0.057,Y -534.237,Z 373.000,A 0.000,B 0.000,C 90.000,E1 35.931} C_DIS
LIN {X 0.144,Y -531.578,Z 372.989,A 0.000,B 0.000,C 90.000,E1 33.913} C_DIS
LIN {X -0.104,Y -529.366,Z 372.979,A 0.000,B 0.000,C 90.000,E1 32.212} C_DIS
LIN {X 0.052,Y -527.240,Z 372.969,A 0.000,B 0.000,C 90.000,E1 30.463} C_DIS
LIN {X 0.037,Y -524.875,Z 372.958,A 0.000,B 0.000,C 90.000,E1 28.437} C_DIS
LIN {X 0.106,Y -522.288,Z 372.945,A 0.000,B 0.000,C 90.000,E1 26.104} C_DIS
LIN {X -0.190,Y -520.473,Z 372.935,A 0.000,B 0.000,C 90.000,E1 24.387} C_DIS
LIN {X 0.069,Y -519.083,Z 372.927,A 0.000,B 0.000,C 90.000,E1 22.898} C_DIS
LIN {X 0.189,Y -516.868,Z 372.913,A 0.000,B 0.000,C 90.000,E1 20.248} C_DIS
LIN {X -0.122,Y -515.104,Z 372.898,A 0.000,B 0.000,C 90.000,E1 17.638} C_DIS
LIN {X 0.184,Y -513.832,Z 372.883,A 0.000,B 0.000,C 90.000,E1 14.954} C_DIS
LIN {X 0.215,Y -513.164,Z 372.870,A 0.000,B 0.000,C 90.000,E1 12.591} C_DIS
LIN {X -0.081,Y -512.986,Z 372.852,A 0.000,B 0.000,C 90.000,E1 9.378} C_DIS
LIN {X 0.031,Y -513.435,Z 372.839,A 0.000,B 0.000,C 90.000,E1 7.004} C_DIS
LIN {X -0.042,Y -514.578,Z 372.824,A 0.000,B 0.000,C 90.000,E1 4.359} C_DIS
LIN {X -0.110,Y -516.481,Z 372.810,A 0.000,B 0.000,C 90.000,E1 1.718} C_DIS
LIN {X -0.131,Y -520.563,Z 372.789,A 0.000,B 0.000,C 90.000,E1 358.051} C_DIS
LIN {X -0.001,Y -524.402,Z 372.775,A 0.000,B 0.000,C 90.000,E1 355.412} C_DIS
LIN {X -0.115,Y -527.929,Z 372.763,A 0.000,B 0.000,C 90.000,E1 353.394} C_DIS
LIN {X -0.062,Y -533.031,Z 372.749,A 0.000,B 0.000,C 90.000,E1 350.792} C_DIS
LIN {X 0.006,Y -541.178,Z 372.730,A 0.000,B 0.000,C 90.000,E1 347.353} C_DIS
LIN {X 0.166,Y -546.654,Z 372.719,A 0.000,B 0.000,C 90.000,E1 345.353} C_DIS
LIN {X -0.198,Y -553.263,Z 372.706,A 0.000,B 0.000,C 90.000,E1 343.142} C_DIS
LIN {X 0.207,Y -559.105,Z 372.695,A 0.000,B 0.000,C 90.000,E1 341.148} C_DIS
LIN {X 0.231,Y -565.046,Z 372.685,A 0.000,B 0.000,C 90.000,E1 339.209} C_DIS
LIN {X 0.111,Y -569.215,Z 372.677,A 0.000,B 0.000,C 90.000,E1 337.847} C_DIS
LIN {X 0.064,Y -573.421,Z 372.669,A 0.000,B 0.000,C 90.000,E1 336.485} C_DIS
LIN {X 0.169,Y -578.467,Z 372.660,A 0.000,B 0.000,C 90.000,E1 334.845} C_DIS
LIN {X 0.263,Y -580.929,Z 372.656,A 0.000,B 0.000,C 90.000,E1 334.024} C_DIS
LIN {X 0.265,Y -586.232,Z 372.647,A 0.000,B 0.000,C 90.000,E1 332.410} C_DIS
LIN {X -0.245,Y -592.548,Z 372.637,A 0.000,B 0.000,C 90.000,E1 330.589} C_DIS
LIN {X -0.235,Y -597.991,Z 372.628,A 0.000,B 0.000,C 90.000,E1 328.997} C_DIS
LIN {X -0.040,Y -602.477,Z 372.620,A 0.000,B 0.000,C 90.000,E1 327.661} C_DIS
LIN {X -0.123,Y -611.579,Z 372.606,A 0.000,B 0.000,C 90.000,E1 325.055} C_DIS
LIN {X -0.016,Y -616.285,Z 372.599,A 0.000,B 0.000,C 90.000,E1 323.749} C_DIS
LIN {X -0.187,Y -621.088,Z 372.591,A 0.000,B 0.000,C 90.000,E1 322.477} C_DIS
LIN {X -0.247,Y -628.750,Z 372.580,A 0.000,B 0.000,C 90.000,E1 320.436} C_DIS
LIN {X -0.084,Y -635.520,Z 372.570,A 0.000,B 0.000,C 90.000,E1 318.647} C_DIS
LIN {X -0.021,Y -639.128,Z 372.565,A 0.000,B 0.000,C 90.000,E1 317.634} C_DIS
LIN {X -0.065,Y -644.468,Z 372.556,A 0.000,B 0.000,C 90.000,E1 316.134} C_DIS
LIN {X 0.054,Y -649.062,Z 372.549,A 0.000,B 0.000,C 90.000,E1 314.879} C_DIS
LIN {X 0.206,Y -654.639,Z 372.541,A 0.000,B 0.000,C 90.000,E1 313.380} C_DIS
LIN {X 0.029,Y -659.950,Z 372.533,A 0.000,B 0.000,C 90.000,E1 311.919} C_DIS
LIN {X -0.046,Y -665.239,Z 372.525,A 0.000,B 0.000,C 90.000,E1 310.458} C_DIS
LIN {X -0.018,Y -668.558,Z 372.519,A 0.000,B 0.000,C 90.000,E1 309.483} C_DIS
LIN {X 0.151,Y -673.451,Z 372.511,A 0.000,B 0.000,C 90.000,E1 308.016} C_DIS
LIN {X -0.137,Y -676.556,Z 372.506,A 0.000,B 0.000,C 90.000,E1 307.076} C_DIS
LIN {X -0.395,Y -678.785,Z 372.502,A 0.000,B 0.000,C 90.000,E1 306.377} C_DIS
LIN {X 0.322,Y -680.830,Z 372.498,A 0.000,B 0.000,C 90.000,E1 305.598} C_DIS
LIN {X 0.297,Y -684.100,Z 372.491,A 0.000,B 0.000,C 90.000,E1 304.405} C_DIS
LIN {X -0.263,Y -686.280,Z 372.486,A 0.000,B 0.000,C 90.000,E1 303.499} C_DIS
LIN {X -0.225,Y -688.182,Z 372.481,A 0.000,B 0.000,C 90.000,E1 302.546} C_DIS
LIN {X 0.204,Y -689.659,Z 372.477,A 0.000,B 0.000,C 90.000,E1 301.799} C_DIS
LIN {X -0.305,Y -690.989,Z 372.473,A 0.000,B 0.000,C 90.000,E1 301.131} C_DIS
LIN {X 0.146,Y -692.042,Z 372.469,A 0.000,B 0.000,C 90.000,E1 300.384} C_DIS
LIN {X 0.257,Y -692.877,Z 372.465,A 0.000,B 0.000,C 90.000,E1 299.667} C_DIS
LIN {X -0.226,Y -693.447,Z 372.461,A 0.000,B 0.000,C 90.000,E1 298.999} C_DIS
LIN {X 0.146,Y -693.599,Z 372.456,A 0.000,B 0.000,C 90.000,E1 298.025} C_DIS
LIN {X -0.295,Y -693.502,Z 372.453,A 0.000,B 0.000,C 90.000,E1 297.590} C_DIS
LIN {X 0.203,Y -693.235,Z 372.451,A 0.000,B 0.000,C 90.000,E1 297.078} C_DIS
LIN {X -0.108,Y -692.017,Z 372.444,A 0.000,B 0.000,C 90.000,E1 295.924} C_DIS
LIN {X -0.004,Y -691.213,Z 372.440,A 0.000,B 0.000,C 90.000,E1 295.207} C_DIS
LIN {X 0.027,Y -689.709,Z 372.435,A 0.000,B 0.000,C 90.000,E1 294.259} C_DIS
LIN {X -0.191,Y -688.519,Z 372.431,A 0.000,B 0.000,C 90.000,E1 293.567} C_DIS
LIN {X -0.252,Y -686.203,Z 372.424,A 0.000,B 0.000,C 90.000,E1 292.386} C_DIS
LIN {X 0.036,Y -683.538,Z 372.418,A 0.000,B 0.000,C 90.000,E1 291.173} C_DIS
LIN {X -0.023,Y -679.192,Z 372.407,A 0.000,B 0.000,C 90.000,E1 289.268} C_DIS
LIN {X 0.105,Y -675.820,Z 372.399,A 0.000,B 0.000,C 90.000,E1 287.819} C_DIS
LIN {X 0.096,Y -672.082,Z 372.390,A 0.000,B 0.000,C 90.000,E1 286.134} C_DIS
LIN {X -0.363,Y -668.411,Z 372.380,A 0.000,B 0.000,C 90.000,E1 284.481} C_DIS
LIN {X 0.156,Y -663.869,Z 372.367,A 0.000,B 0.000,C 90.000,E1 282.007} C_DIS
LIN {X -0.292,Y -658.800,Z 372.348,A 0.000,B 0.000,C 90.000,E1 278.624} C_DIS
LIN {X -0.036,Y -655.554,Z 372.329,A 0.000,B 0.000,C 90.000,E1 275.163} C_DIS
LIN {X 0.245,Y -654.425,Z 372.316,A 0.000,B 0.000,C 90.000,E1 272.922} C_DIS
LIN {X 0.230,Y -653.898,Z 372.303,A 0.000,B 0.000,C 90.000,E1 270.458} C_DIS
LIN {X 0.016,Y -654.118,Z 372.288,A 0.000,B 0.000,C 90.000,E1 267.764} C_DIS
LIN {X 0.239,Y -654.969,Z 372.275,A 0.000,B 0.000,C 90.000,E1 265.527} C_DIS
LIN {X -0.230,Y -655.544,Z 372.267,A 0.000,B 0.000,C 90.000,E1 264.090} C_DIS
LIN {X 0.240,Y -655.719,Z 372.260,A 0.000,B 0.000,C 90.000,E1 262.818} C_DIS
LIN {X -0.105,Y -655.725,Z 372.258,A 0.000,B 0.000,C 90.000,E1 262.356} C_DIS
LIN {X 0.198,Y -655.687,Z 372.255,A 0.000,B 0.000,C 90.000,E1 261.837} C_DIS
LIN {X 0.071,Y -655.573,Z 372.253,A 0.000,B 0.000,C 90.000,E1 261.602} C_DIS
LIN {X -0.151,Y -655.640,Z 372.252,A 0.000,B 0.000,C 90.000,E1 261.376} C_DIS
LIN {X 0.019,Y -655.205,Z 372.248,A 0.000,B 0.000,C 90.000,E1 260.622} C_DIS
LIN {X -0.181,Y -654.083,Z 372.240,A 0.000,B 0.000,C 90.000,E1 259.162} C_DIS
LIN {X -0.153,Y -653.395,Z 372.234,A 0.000,B 0.000,C 90.000,E1 258.173} C_DIS
LIN {X 0.120,Y -652.682,Z 372.230,A 0.000,B 0.000,C 90.000,E1 257.409} C_DIS
LIN {X 0.137,Y -650.951,Z 372.223,A 0.000,B 0.000,C 90.000,E1 256.172} C_DIS
LIN {X -0.246,Y -649.786,Z 372.219,A 0.000,B 0.000,C 90.000,E1 255.463} C_DIS
LIN {X -0.112,Y -647.248,Z 372.212,A 0.000,B 0.000,C 90.000,E1 254.212} C_DIS
LIN {X 0.085,Y -645.420,Z 372.208,A 0.000,B 0.000,C 90.000,E1 253.449} C_DIS
LIN {X -0.174,Y -643.362,Z 372.204,A 0.000,B 0.000,C 90.000,E1 252.725} C_DIS
LIN {X 0.202,Y -640.365,Z 372.198,A 0.000,B 0.000,C 90.000,E1 251.692} C_DIS
LIN {X -0.272,Y -637.020,Z 372.193,A 0.000,B 0.000,C 90.000,E1 250.732} C_DIS
LIN {X 0.017,Y -633.251,Z 372.187,A 0.000,B 0.000,C 90.000,E1 249.699} C_DIS
LIN {X 0.263,Y -628.408,Z 372.180,A 0.000,B 0.000,C 90.000,E1 248.411} C_DIS
LIN {X -0.158,Y -623.369,Z 372.173,A 0.000,B 0.000,C 90.000,E1 247.177} C_DIS
LIN {X 0.137,Y -616.981,Z 372.165,A 0.000,B 0.000,C 90.000,E1 245.613} C_DIS
LIN {X 0.061,Y -612.636,Z 372.159,A 0.000,B 0.000,C 90.000,E1 244.588} C_DIS
LIN {X -0.195,Y -605.054,Z 372.149,A 0.000,B 0.000,C 90.000,E1 242.794} C_DIS
LIN {X 0.038,Y -599.700,Z 372.142,A 0.000,B 0.000,C 90.000,E1 241.463} C_DIS
LIN {X 0.219,Y -594.333,Z 372.134,A 0.000,B 0.000,C 90.000,E1 240.127} C_DIS
LIN {X 0.270,Y -586.042,Z 372.122,A 0.000,B 0.000,C 90.000,E1 237.995} C_DIS
LIN {X 0.069,Y -577.362,Z 372.109,A 0.000,B 0.000,C 90.000,E1 235.595} C_DIS
LIN {X -0.155,Y -571.917,Z 372.100,A 0.000,B 0.000,C 90.000,E1 233.989} C_DIS
LIN {X -0.283,Y -567.388,Z 372.092,A 0.000,B 0.000,C 90.000,E1 232.637} C_DIS
LIN {X -0.256,Y -563.625,Z 372.086,A 0.000,B 0.000,C 90.000,E1 231.537} C_DIS
LIN {X -0.084,Y -556.886,Z 372.075,A 0.000,B 0.000,C 90.000,E1 229.585} C_DIS
LIN {X 0.335,Y -549.530,Z 372.063,A 0.000,B 0.000,C 90.000,E1 227.310} C_DIS
LIN {X 0.083,Y -544.112,Z 372.054,A 0.000,B 0.000,C 90.000,E1 225.648} C_DIS
LIN {X 0.097,Y -538.700,Z 372.044,A 0.000,B 0.000,C 90.000,E1 223.947} C_DIS
LIN {X -0.036,Y -532.516,Z 372.033,A 0.000,B 0.000,C 90.000,E1 221.962} C_DIS
LIN {X 0.076,Y -525.616,Z 372.020,A 0.000,B 0.000,C 90.000,E1 219.644} C_DIS
LIN {X 0.127,Y -519.799,Z 372.009,A 0.000,B 0.000,C 90.000,E1 217.604} C_DIS
LIN {X -0.211,Y -515.054,Z 371.999,A 0.000,B 0.000,C 90.000,E1 215.884} C_DIS
LIN {X 0.095,Y -509.694,Z 371.988,A 0.000,B 0.000,C 90.000,E1 213.785} C_DIS
LIN {X 0.079,Y -505.383,Z 371.978,A 0.000,B 0.000,C 90.000,E1 212.005} C_DIS
LIN {X -0.173,Y -501.916,Z 371.970,A 0.000,B 0.000,C 90.000,E1 210.541} C_DIS
LIN {X -0.199,Y -497.830,Z 371.960,A 0.000,B 0.000,C 90.000,E1 208.743} C_DIS
LIN {X -0.094,Y -493.079,Z 371.948,A 0.000,B 0.000,C 90.000,E1 206.616} C_DIS
LIN {X 0.057,Y -489.619,Z 371.939,A 0.000,B 0.000,C 90.000,E1 205.079} C_DIS
LIN {X -0.070,Y -486.060,Z 371.931,A 0.000,B 0.000,C 90.000,E1 203.567} C_DIS
LIN {X -0.002,Y -481.692,Z 371.921,A 0.000,B 0.000,C 90.000,E1 201.716} C_DIS
LIN {X -0.215,Y -476.617,Z 371.909,A 0.000,B 0.000,C 90.000,E1 199.577} C_DIS
LIN {X -0.264,Y -471.803,Z 371.897,A 0.000,B 0.000,C 90.000,E1 197.402} C_DIS
LIN {X 0.057,Y -467.870,Z 371.886,A 0.000,B 0.000,C 90.000,E1 195.481} C_DIS
LIN {X 0.034,Y -464.144,Z 371.876,A 0.000,B 0.000,C 90.000,E1 193.592} C_DIS
LIN {X -0.142,Y -459.472,Z 371.861,A 0.000,B 0.000,C 90.000,E1 191.074} C_DIS
LIN {X 0.133,Y -455.622,Z 371.849,A 0.000,B 0.000,C 90.000,E1 188.803} C_DIS
LIN {X 0.118,Y -451.051,Z 371.833,A 0.000,B 0.000,C 90.000,E1 185.910} C_DIS
LIN {X 0.077,Y -447.522,Z 371.819,A 0.000,B 0.000,C 90.000,E1 183.326} C_DIS
LIN {X -0.087,Y -444.713,Z 371.804,A 0.000,B 0.000,C 90.000,E1 180.745} C_DIS
LIN {X -0.089,Y -442.230,Z 371.786,A 0.000,B 0.000,C 90.000,E1 177.478} C_DIS
LIN {X -0.187,Y -440.372,Z 371.757,A 0.000,B 0.000,C 90.000,E1 172.243} C_DIS
LIN {X 0.061,Y -440.645,Z 371.739,A 0.000,B 0.000,C 90.000,E1 168.926} C_DIS
LIN {X 0.070,Y -442.128,Z 371.720,A 0.000,B 0.000,C 90.000,E1 165.644} C_DIS
LIN {X 0.155,Y -444.827,Z 371.702,A 0.000,B 0.000,C 90.000,E1 162.362} C_DIS
LIN {X 0.057,Y -448.082,Z 371.686,A 0.000,B 0.000,C 90.000,E1 159.444} C_DIS
LIN {X -0.078,Y -451.782,Z 371.671,A 0.000,B 0.000,C 90.000,E1 156.869} C_DIS
LIN {X -0.089,Y -456.645,Z 371.655,A 0.000,B 0.000,C 90.000,E1 153.973} C_DIS
LIN {X -0.213,Y -463.189,Z 371.638,A 0.000,B 0.000,C 90.000,E1 150.795} C_DIS
LIN {X 0.166,Y -472.778,Z 371.617,A 0.000,B 0.000,C 90.000,E1 146.962} C_DIS
LIN {X 0.154,Y -483.317,Z 371.598,A 0.000,B 0.000,C 90.000,E1 143.543} C_DIS
LIN {X -0.048,Y -488.550,Z 371.589,A 0.000,B 0.000,C 90.000,E1 142.029} C_DIS
LIN {X -0.162,Y -493.741,Z 371.581,A 0.000,B 0.000,C 90.000,E1 140.517} C_DIS
LIN {X -0.114,Y -497.766,Z 371.574,A 0.000,B 0.000,C 90.000,E1 139.299} C_DIS
LIN {X -0.001,Y -501.714,Z 371.567,A 0.000,B 0.000,C 90.000,E1 138.081} C_DIS
LIN {X 0.166,Y -505.412,Z 371.561,A 0.000,B 0.000,C 90.000,E1 136.863} C_DIS
LIN {X 0.132,Y -508.045,Z 371.556,A 0.000,B 0.000,C 90.000,E1 135.972} C_DIS
LIN {X 0.014,Y -511.201,Z 371.549,A 0.000,B 0.000,C 90.000,E1 134.798} C_DIS
LIN {X -0.315,Y -513.350,Z 371.544,A 0.000,B 0.000,C 90.000,E1 133.947} C_DIS
LIN {X 0.203,Y -514.604,Z 371.541,A 0.000,B 0.000,C 90.000,E1 133.299} C_DIS
LIN {X 0.001,Y -515.792,Z 371.537,A 0.000,B 0.000,C 90.000,E1 132.732} C_DIS
LIN {X 0.108,Y -517.337,Z 371.533,A 0.000,B 0.000,C 90.000,E1 131.838} C_DIS
LIN {X -0.150,Y -518.559,Z 371.528,A 0.000,B 0.000,C 90.000,E1 130.987} C_DIS
LIN {X -0.063,Y -519.679,Z 371.521,A 0.000,B 0.000,C 90.000,E1 129.806} C_DIS
LIN {X 0.100,Y -520.013,Z 371.516,A 0.000,B 0.000,C 90.000,E1 128.910} C_DIS
LIN {X -0.006,Y -520.004,Z 371.513,A 0.000,B 0.000,C 90.000,E1 128.338} C_DIS
LIN {X 0.208,Y -519.792,Z 371.510,A 0.000,B 0.000,C 90.000,E1 127.729} C_DIS
LIN {X 0.048,Y -519.211,Z 371.505,A 0.000,B 0.000,C 90.000,E1 126.870} C_DIS
LIN {X -0.118,Y -518.391,Z 371.500,A 0.000,B 0.000,C 90.000,E1 126.011} C_DIS
LIN {X 0.126,Y -517.245,Z 371.495,A 0.000,B 0.000,C 90.000,E1 125.105} C_DIS
LIN {X -0.068,Y -515.873,Z 371.490,A 0.000,B 0.000,C 90.000,E1 124.246} C_DIS
LIN {X -0.140,Y -514.266,Z 371.485,A 0.000,B 0.000,C 90.000,E1 123.372} C_DIS
LIN {X -0.305,Y -511.829,Z 371.479,A 0.000,B 0.000,C 90.000,E1 122.212} C_DIS
LIN {X -0.051,Y -510.361,Z 371.476,A 0.000,B 0.000,C 90.000,E1 121.592} C_DIS
LIN {X -0.219,Y -506.280,Z 371.467,A 0.000,B 0.000,C 90.000,E1 120.129} C_DIS
LIN {X 0.045,Y -503.568,Z 371.462,A 0.000,B 0.000,C 90.000,E1 119.205} C_DIS
LIN {X 0.037,Y -500.582,Z 371.457,A 0.000,B 0.000,C 90.000,E1 118.309} C_DIS
LIN {X 0.233,Y -497.285,Z 371.452,A 0.000,B 0.000,C 90.000,E1 117.385} C_DIS
LIN {X 0.114,Y -495.100,Z 371.449,A 0.000,B 0.000,C 90.000,E1 116.796} C_DIS
LIN {X 0.046,Y -490.330,Z 371.442,A 0.000,B 0.000,C 90.000,E1 115.591} C_DIS
LIN {X 0.119,Y -485.861,Z 371.436,A 0.000,B 0.000,C 90.000,E1 114.515} C_DIS
LIN {X -0.288,Y -480.444,Z 371.430,A 0.000,B 0.000,C 90.000,E1 113.334} C_DIS
LIN {X -0.126,Y -476.189,Z 371.424,A 0.000,B 0.000,C 90.000,E1 112.386} C_DIS
LIN {X 0.004,Y -471.000,Z 371.418,A 0.000,B 0.000,C 90.000,E1 111.280} C_DIS
LIN {X 0.030,Y -463.330,Z 371.410,A 0.000,B 0.000,C 90.000,E1 109.704} C_DIS
LIN {X -0.108,Y -459.103,Z 371.405,A 0.000,B 0.000,C 90.000,E1 108.833} C_DIS
LIN {X -0.148,Y -459.090,Z 371.405,A 0.000,B 0.000,C 90.000,E1 108.833} C_DIS
LIN {X -0.083,Y -467.667,Z 371.383,A 0.000,B 0.000,C 90.000,E1 104.954} C_DIS
LIN {X -0.094,Y -473.980,Z 371.362,A 0.000,B 0.000,C 90.000,E1 101.186} C_DIS
LIN {X -0.125,Y -475.882,Z 371.357,A 0.000,B 0.000,C 90.000,E1 100.254} C_DIS
LIN {X 0.182,Y -476.341,Z 371.355,A 0.000,B 0.000,C 90.000,E1 99.905} C_DIS
LIN {X 0.139,Y -481.850,Z 371.331,A 0.000,B 0.000,C 90.000,E1 95.568} C_DIS
LIN {X -0.014,Y -482.187,Z 371.329,A 0.000,B 0.000,C 90.000,E1 95.277} C_DIS
LIN {X -0.080,Y -485.348,Z 371.305,A 0.000,B 0.000,C 90.000,E1 90.974} C_DIS
LIN {X 0.230,Y -485.533,Z 371.304,A 0.000,B 0.000,C 90.000,E1 90.630} C_DIS
LIN {X -0.048,Y -486.338,Z 371.282,A 0.000,B 0.000,C 90.000,E1 86.674} C_DIS
LIN {X 0.087,Y -486.278,Z 371.278,A 0.000,B 0.000,C 90.000,E1 86.045} C_DIS
LIN {X -0.194,Y -484.694,Z 371.254,A 0.000,B 0.000,C 90.000,E1 81.781} C_DIS
LIN {X 0.154,Y -484.553,Z 371.253,A 0.000,B 0.000,C 90.000,E1 81.432} C_DIS
LIN {X 0.024,Y -480.493,Z 371.227,A 0.000,B 0.000,C 90.000,E1 76.825} C_DIS
LIN {X 0.129,Y -475.029,Z 371.205,A 0.000,B 0.000,C 90.000,E1 72.906} C_DIS
LIN {X 0.089,Y -475.052,Z 371.205,A 0.000,B 0.000,C 90.000,E1 72.906} C_DIS
LIN {X -0.248,Y -484.204,Z 371.198,A 0.000,B 0.000,C 90.000,E1 71.583} C_DIS
LIN {X -0.142,Y -491.093,Z 371.192,A 0.000,B 0.000,C 90.000,E1 70.496} C_DIS
LIN {X 0.135,Y -493.820,Z 371.189,A 0.000,B 0.000,C 90.000,E1 70.007} C_DIS
LIN {X -0.141,Y -496.492,Z 371.187,A 0.000,B 0.000,C 90.000,E1 69.625} C_DIS
LIN {X 0.076,Y -500.865,Z 371.183,A 0.000,B 0.000,C 90.000,E1 68.847} C_DIS
LIN {X -0.247,Y -503.829,Z 371.179,A 0.000,B 0.000,C 90.000,E1 68.284} C_DIS
LIN {X 0.116,Y -505.949,Z 371.177,A 0.000,B 0.000,C 90.000,E1 67.847} C_DIS
LIN {X -0.314,Y -507.915,Z 371.175,A 0.000,B 0.000,C 90.000,E1 67.486} C_DIS
LIN {X -0.098,Y -511.439,Z 371.171,A 0.000,B 0.000,C 90.000,E1 66.719} C_DIS
LIN {X -0.046,Y -514.647,Z 371.167,A 0.000,B 0.000,C 90.000,E1 65.973} C_DIS
LIN {X 0.201,Y -516.988,Z 371.163,A 0.000,B 0.000,C 90.000,E1 65.357} C_DIS
LIN {X 0.124,Y -520.003,Z 371.158,A 0.000,B 0.000,C 90.000,E1 64.485} C_DIS
LIN {X -0.020,Y -523.743,Z 371.152,A 0.000,B 0.000,C 90.000,E1 63.332} C_DIS
LIN {X -0.176,Y -527.947,Z 371.144,A 0.000,B 0.000,C 90.000,E1 61.897} C_DIS
LIN {X 0.049,Y -531.250,Z 371.137,A 0.000,B 0.000,C 90.000,E1 60.717} C_DIS
LIN {X 0.030,Y -535.186,Z 371.129,A 0.000,B 0.000,C 90.000,E1 59.282} C_DIS
LIN {X 0.172,Y -538.203,Z 371.123,A 0.000,B 0.000,C 90.000,E1 58.122} C_DIS
LIN {X 0.072,Y -540.992,Z 371.117,A 0.000,B 0.000,C 90.000,E1 56.993} C_DIS
LIN {X -0.151,Y -543.707,Z 371.110,A 0.000,B 0.000,C 90.000,E1 55.881} C_DIS
LIN {X -0.057,Y -545.565,Z 371.106,A 0.000,B 0.000,C 90.000,E1 55.022} C_DIS
LIN {X -0.212,Y -547.744,Z 371.099,A 0.000,B 0.000,C 90.000,E1 53.909} C_DIS
LIN {X -0.118,Y -548.694,Z 371.096,A 0.000,B 0.000,C 90.000,E1 53.336} C_DIS
LIN {X 0.038,Y -549.832,Z 371.092,A 0.000,B 0.000,C 90.000,E1 52.477} C_DIS
LIN {X 0.203,Y -550.708,Z 371.087,A 0.000,B 0.000,C 90.000,E1 51.618} C_DIS
LIN {X -0.056,Y -551.284,Z 371.082,A 0.000,B 0.000,C 90.000,E1 50.803} C_DIS
LIN {X -0.308,Y -551.349,Z 371.078,A 0.000,B 0.000,C 90.000,E1 49.989} C_DIS
LIN {X 0.214,Y -551.342,Z 371.073,A 0.000,B 0.000,C 90.000,E1 49.094} C_DIS
LIN {X 0.320,Y -550.951,Z 371.068,A 0.000,B 0.000,C 90.000,E1 48.243} C_DIS
LIN {X 0.063,Y -550.027,Z 371.062,A 0.000,B 0.000,C 90.000,E1 47.148} C_DIS
LIN {X 0.158,Y -549.059,Z 371.057,A 0.000,B 0.000,C 90.000,E1 46.296} C_DIS
LIN {X -0.074,Y -546.378,Z 371.046,A 0.000,B 0.000,C 90.000,E1 44.352} C_DIS
LIN {X -0.373,Y -544.057,Z 371.037,A 0.000,B 0.000,C 90.000,E1 42.690} C_DIS
LIN {X -0.305,Y -541.366,Z 371.026,A 0.000,B 0.000,C 90.000,E1 40.701} C_DIS
LIN {X 0.084,Y -539.106,Z 371.017,A 0.000,B 0.000,C 90.000,E1 38.955} C_DIS
LIN {X 0.153,Y -537.243,Z 371.009,A 0.000,B 0.000,C 90.000,E1 37.523} C_DIS
LIN {X 0.194,Y -535.391,Z 371.001,A 0.000,B 0.000,C 90.000,E1 36.091} C_DIS
LIN {X -0.115,Y -533.093,Z 370.991,A 0.000,B 0.000,C 90.000,E1 34.405} C_DIS
LIN {X -0.059,Y -530.522,Z 370.980,A 0.000,B 0.000,C 90.000,E1 32.388} C_DIS
LIN {X -0.160,Y -528.400,Z 370.970,A 0.000,B 0.000,C 90.000,E1 30.669} C_DIS
LIN {X 0.112,Y -526.061,Z 370.959,A 0.000,B 0.000,C 90.000,E1 28.615} C_DIS
LIN {X -0.112,Y -523.162,Z 370.945,A 0.000,B 0.000,C 90.000,E1 26.027} C_DIS
LIN {X 0.080,Y -521.361,Z 370.935,A 0.000,B 0.000,C 90.000,E1 24.259} C_DIS
LIN {X -0.125,Y -519.972,Z 370.927,A 0.000,B 0.000,C 90.000,E1 22.823} C_DIS
LIN {X 0.012,Y -517.796,Z 370.912,A 0.000,B 0.000,C 90.000,E1 20.174} C_DIS
LIN {X 0.209,Y -516.056,Z 370.897,A 0.000,B 0.000,C 90.000,E1 17.511} C_DIS
LIN {X -0.068,Y -514.961,Z 370.884,A 0.000,B 0.000,C 90.000,E1 15.190} C_DIS
LIN {X -0.026,Y -514.222,Z 370.870,A 0.000,B 0.000,C 90.000,E1 12.535} C_DIS
LIN {X -0.248,Y -514.084,Z 370.853,A 0.000,B 0.000,C 90.000,E1 9.613} C_DIS
LIN {X -0.094,Y -514.520,Z 370.840,A 0.000,B 0.000,C 90.000,E1 7.239} C_DIS
LIN {X -0.044,Y -515.472,Z 370.827,A 0.000,B 0.000,C 90.000,E1 4.878} C_DIS
LIN {X -0.069,Y -517.261,Z 370.812,A 0.000,B 0.000,C 90.000,E1 2.236} C_DIS
LIN {X -0.070,Y -521.490,Z 370.791,A 0.000,B 0.000,C 90.000,E1 358.339} C_DIS
LIN {X 0.072,Y -526.223,Z 370.773,A 0.000,B 0.000,C 90.000,E1 355.122} C_DIS
LIN {X -0.022,Y -530.367,Z 370.760,A 0.000,B 0.000,C 90.000,E1 352.818} C_DIS
LIN {X 0.209,Y -536.949,Z 370.743,A 0.000,B 0.000,C 90.000,E1 349.634} C_DIS
LIN {X -0.230,Y -543.276,Z 370.728,A 0.000,B 0.000,C 90.000,E1 347.117} C_DIS
LIN {X -0.202,Y -547.252,Z 370.720,A 0.000,B 0.000,C 90.000,E1 345.700} C_DIS
LIN {X -0.012,Y -553.817,Z 370.708,A 0.000,B 0.000,C 90.000,E1 343.433} C_DIS
LIN {X -0.055,Y -558.808,Z 370.699,A 0.000,B 0.000,C 90.000,E1 341.764} C_DIS
LIN {X 0.040,Y -563.065,Z 370.691,A 0.000,B 0.000,C 90.000,E1 340.369} C_DIS
LIN {X -0.323,Y -567.355,Z 370.683,A 0.000,B 0.000,C 90.000,E1 339.028} C_DIS
LIN {X -0.229,Y -573.220,Z 370.673,A 0.000,B 0.000,C 90.000,E1 337.102} C_DIS
LIN {X 0.011,Y -579.119,Z 370.662,A 0.000,B 0.000,C 90.000,E1 335.177} C_DIS
LIN {X 0.112,Y -586.851,Z 370.649,A 0.000,B 0.000,C 90.000,E1 332.743} C_DIS
LIN {X -0.179,Y -591.341,Z 370.641,A 0.000,B 0.000,C 90.000,E1 331.435} C_DIS
LIN {X 0.123,Y -595.883,Z 370.634,A 0.000,B 0.000,C 90.000,E1 330.078} C_DIS
LIN {X -0.318,Y -601.344,Z 370.625,A 0.000,B 0.000,C 90.000,E1 328.535} C_DIS
LIN {X 0.258,Y -605.759,Z 370.618,A 0.000,B 0.000,C 90.000,E1 327.168} C_DIS
LIN {X 0.067,Y -613.119,Z 370.606,A 0.000,B 0.000,C 90.000,E1 325.102} C_DIS
LIN {X -0.155,Y -617.813,Z 370.599,A 0.000,B 0.000,C 90.000,E1 323.829} C_DIS
LIN {X -0.304,Y -622.616,Z 370.592,A 0.000,B 0.000,C 90.000,E1 322.557} C_DIS
LIN {X 0.208,Y -629.297,Z 370.582,A 0.000,B 0.000,C 90.000,E1 320.723} C_DIS
LIN {X 0.290,Y -636.998,Z 370.571,A 0.000,B 0.000,C 90.000,E1 318.690} C_DIS
LIN {X -0.049,Y -640.590,Z 370.565,A 0.000,B 0.000,C 90.000,E1 317.715} C_DIS
LIN {X -0.201,Y -647.758,Z 370.554,A 0.000,B 0.000,C 90.000,E1 315.729} C_DIS
LIN {X 0.341,Y -654.188,Z 370.544,A 0.000,B 0.000,C 90.000,E1 313.947} C_DIS
LIN {X 0.220,Y -656.952,Z 370.540,A 0.000,B 0.000,C 90.000,E1 313.218} C_DIS
LIN {X 0.064,Y -663.080,Z 370.531,A 0.000,B 0.000,C 90.000,E1 311.515} C_DIS
LIN {X 0.052,Y -667.427,Z 370.524,A 0.000,B 0.000,C 90.000,E1 310.297} C_DIS
LIN {X -0.223,Y -673.091,Z 370.515,A 0.000,B 0.000,C 90.000,E1 308.624} C_DIS
LIN {X -0.098,Y -676.277,Z 370.509,A 0.000,B 0.000,C 90.000,E1 307.649} C_DIS
LIN {X 0.191,Y -679.326,Z 370.504,A 0.000,B 0.000,C 90.000,E1 306.664} C_DIS
LIN {X -0.026,Y -682.028,Z 370.499,A 0.000,B 0.000,C 90.000,E1 305.724} C_DIS
LIN {X -0.038,Y -685.253,Z 370.492,A 0.000,B 0.000,C 90.000,E1 304.532} C_DIS
LIN {X -0.214,Y -686.900,Z 370.488,A 0.000,B 0.000,C 90.000,E1 303.833} C_DIS
LIN {X -0.386,Y -687.905,Z 370.485,A 0.000,B 0.000,C 90.000,E1 303.372} C_DIS
LIN {X 0.120,Y -690.908,Z 370.476,A 0.000,B 0.000,C 90.000,E1 301.671} C_DIS
LIN {X -0.014,Y -691.711,Z 370.473,A 0.000,B 0.000,C 90.000,E1 301.209} C_DIS
LIN {X -0.148,Y -692.606,Z 370.469,A 0.000,B 0.000,C 90.000,E1 300.512} C_DIS
LIN {X -0.033,Y -693.297,Z 370.466,A 0.000,B 0.000,C 90.000,E1 299.795} C_DIS
LIN {X 0.092,Y -693.704,Z 370.462,A 0.000,B 0.000,C 90.000,E1 299.077} C_DIS
LIN {X -0.128,Y -693.671,Z 370.456,A 0.000,B 0.000,C 90.000,E1 298.153} C_DIS
LIN {X 0.119,Y -693.668,Z 370.455,A 0.000,B 0.000,C 90.000,E1 297.897} C_DIS
LIN {X -0.071,Y -693.280,Z 370.451,A 0.000,B 0.000,C 90.000,E1 297.206} C_DIS
LIN {X 0.300,Y -692.255,Z 370.446,A 0.000,B 0.000,C 90.000,E1 296.232} C_DIS
LIN {X -0.276,Y -691.014,Z 370.441,A 0.000,B 0.000,C 90.000,E1 295.335} C_DIS
LIN {X -0.245,Y -689.463,Z 370.435,A 0.000,B 0.000,C 90.000,E1 294.387} C_DIS
LIN {X 0.392,Y -687.637,Z 370.430,A 0.000,B 0.000,C 90.000,E1 293.387} C_DIS
LIN {X 0.318,Y -685.165,Z 370.424,A 0.000,B 0.000,C 90.000,E1 292.206} C_DIS
LIN {X 0.149,Y -681.847,Z 370.416,A 0.000,B 0.000,C 90.000,E1 290.791} C_DIS
LIN {X -0.142,Y -677.960,Z 370.406,A 0.000,B 0.000,C 90.000,E1 289.141} C_DIS
LIN {X -0.158,Y -673.492,Z 370.396,A 0.000,B 0.000,C 90.000,E1 287.221} C_DIS
LIN {X -0.336,Y -670.215,Z 370.388,A 0.000,B 0.000,C 90.000,E1 285.788} C_DIS
LIN {X -0.246,Y -665.210,Z 370.374,A 0.000,B 0.000,C 90.000,E1 283.355} C_DIS
LIN {X 0.018,Y -660.953,Z 370.361,A 0.000,B 0.000,C 90.000,E1 280.894} C_DIS
LIN {X -0.092,Y -657.613,Z 370.347,A 0.000,B 0.000,C 90.000,E1 278.454} C_DIS
LIN {X 0.125,Y -654.447,Z 370.328,A 0.000,B 0.000,C 90.000,E1 274.992} C_DIS
LIN {X -0.276,Y -653.391,Z 370.316,A 0.000,B 0.000,C 90.000,E1 272.808} C_DIS
LIN {X -0.321,Y -652.885,Z 370.302,A 0.000,B 0.000,C 90.000,E1 270.344} C_DIS
LIN {X -0.122,Y -653.308,Z 370.285,A 0.000,B 0.000,C 90.000,E1 267.364} C_DIS
LIN {X -0.172,Y -654.005,Z 370.276,A 0.000,B 0.000,C 90.000,E1 265.641} C_DIS
LIN {X -0.148,Y -654.653,Z 370.266,A 0.000,B 0.000,C 90.000,E1 263.913} C_DIS
LIN {X -0.199,Y -654.896,Z 370.261,A 0.000,B 0.000,C 90.000,E1 262.932} C_DIS
LIN {X -0.248,Y -655.073,Z 370.255,A 0.000,B 0.000,C 90.000,E1 261.951} C_DIS
LIN {X -0.079,Y -655.078,Z 370.251,A 0.000,B 0.000,C 90.000,E1 261.197} C_DIS
LIN {X 0.092,Y -654.814,Z 370.247,A 0.000,B 0.000,C 90.000,E1 260.443} C_DIS
LIN {X 0.014,Y -654.024,Z 370.240,A 0.000,B 0.000,C 90.000,E1 259.218} C_DIS
LIN {X 0.043,Y -653.361,Z 370.235,A 0.000,B 0.000,C 90.000,E1 258.229} C_DIS
LIN {X 0.318,Y -652.737,Z 370.231,A 0.000,B 0.000,C 90.000,E1 257.465} C_DIS
LIN {X 0.340,Y -651.374,Z 370.224,A 0.000,B 0.000,C 90.000,E1 256.228} C_DIS
LIN {X 0.215,Y -650.926,Z 370.222,A 0.000,B 0.000,C 90.000,E1 255.992} C_DIS
LIN {X -0.166,Y -650.021,Z 370.218,A 0.000,B 0.000,C 90.000,E1 255.283} C_DIS
LIN {X -0.026,Y -647.641,Z 370.211,A 0.000,B 0.000,C 90.000,E1 254.031} C_DIS
LIN {X 0.218,Y -645.266,Z 370.206,A 0.000,B 0.000,C 90.000,E1 253.015} C_DIS
LIN {X -0.230,Y -643.256,Z 370.202,A 0.000,B 0.000,C 90.000,E1 252.308} C_DIS
LIN {X 0.104,Y -641.035,Z 370.197,A 0.000,B 0.000,C 90.000,E1 251.529} C_DIS
LIN {X 0.015,Y -638.598,Z 370.193,A 0.000,B 0.000,C 90.000,E1 250.786} C_DIS
LIN {X 0.327,Y -634.878,Z 370.188,A 0.000,B 0.000,C 90.000,E1 249.752} C_DIS
LIN {X -0.214,Y -630.083,Z 370.181,A 0.000,B 0.000,C 90.000,E1 248.539} C_DIS
LIN {X 0.212,Y -625.151,Z 370.174,A 0.000,B 0.000,C 90.000,E1 247.230} C_DIS
LIN {X -0.014,Y -619.858,Z 370.167,A 0.000,B 0.000,C 90.000,E1 245.973} C_DIS
LIN {X 0.233,Y -614.483,Z 370.159,A 0.000,B 0.000,C 90.000,E1 244.665} C_DIS
LIN {X 0.009,Y -606.899,Z 370.149,A 0.000,B 0.000,C 90.000,E1 242.871} C_DIS
LIN {X 0.025,Y -601.567,Z 370.142,A 0.000,B 0.000,C 90.000,E1 241.563} C_DIS
LIN {X -0.045,Y -596.232,Z 370.135,A 0.000,B 0.000,C 90.000,E1 240.255} C_DIS
LIN {X 0.066,Y -587.919,Z 370.123,A 0.000,B 0.000,C 90.000,E1 238.122} C_DIS
LIN {X -0.069,Y -579.209,Z 370.110,A 0.000,B 0.000,C 90.000,E1 235.722} C_DIS
LIN {X -0.100,Y -572.859,Z 370.099,A 0.000,B 0.000,C 90.000,E1 233.829} C_DIS
LIN {X 0.114,Y -569.249,Z 370.093,A 0.000,B 0.000,C 90.000,E1 232.718} C_DIS
LIN {X -0.164,Y -564.528,Z 370.085,A 0.000,B 0.000,C 90.000,E1 231.376} C_DIS
LIN {X 0.118,Y -556.863,Z 370.073,A 0.000,B 0.000,C 90.000,E1 229.138} C_DIS
LIN {X -0.296,Y -550.467,Z 370.062,A 0.000,B 0.000,C 90.000,E1 227.229} C_DIS
LIN {X 0.250,Y -545.043,Z 370.053,A 0.000,B 0.000,C 90.000,E1 225.486} C_DIS
LIN {X -0.097,Y -540.526,Z 370.045,A 0.000,B 0.000,C 90.000,E1 224.109} C_DIS
LIN {X -0.189,Y -533.461,Z 370.032,A 0.000,B 0.000,C 90.000,E1 221.838} C_DIS
LIN {X -0.034,Y -526.548,Z 370.020,A 0.000,B 0.000,C 90.000,E1 219.519} C_DIS
LIN {X 0.320,Y -519.914,Z 370.007,A 0.000,B 0.000,C 90.000,E1 217.156} C_DIS
LIN {X -0.026,Y -515.188,Z 369.997,A 0.000,B 0.000,C 90.000,E1 215.438} C_DIS
LIN {X -0.103,Y -509.145,Z 369.984,A 0.000,B 0.000,C 90.000,E1 213.086} C_DIS
LIN {X 0.083,Y -506.309,Z 369.977,A 0.000,B 0.000,C 90.000,E1 211.878} C_DIS
LIN {X 0.105,Y -502.859,Z 369.969,A 0.000,B 0.000,C 90.000,E1 210.384} C_DIS
LIN {X -0.153,Y -498.792,Z 369.959,A 0.000,B 0.000,C 90.000,E1 208.615} C_DIS
LIN {X -0.023,Y -494.056,Z 369.947,A 0.000,B 0.000,C 90.000,E1 206.488} C_DIS
LIN {X 0.147,Y -490.608,Z 369.939,A 0.000,B 0.000,C 90.000,E1 204.951} C_DIS
LIN {X -0.157,Y -487.089,Z 369.930,A 0.000,B 0.000,C 90.000,E1 203.462} C_DIS
LIN {X 0.124,Y -482.727,Z 369.920,A 0.000,B 0.000,C 90.000,E1 201.589} C_DIS
LIN {X -0.067,Y -477.671,Z 369.908,A 0.000,B 0.000,C 90.000,E1 199.450} C_DIS
LIN {X -0.095,Y -472.881,Z 369.896,A 0.000,B 0.000,C 90.000,E1 197.275} C_DIS
LIN {X 0.057,Y -468.346,Z 369.884,A 0.000,B 0.000,C 90.000,E1 195.064} C_DIS
LIN {X 0.042,Y -464.625,Z 369.873,A 0.000,B 0.000,C 90.000,E1 193.175} C_DIS
LIN {X 0.082,Y -460.599,Z 369.861,A 0.000,B 0.000,C 90.000,E1 190.950} C_DIS
LIN {X -0.146,Y -456.740,Z 369.849,A 0.000,B 0.000,C 90.000,E1 188.746} C_DIS
LIN {X -0.117,Y -452.169,Z 369.832,A 0.000,B 0.000,C 90.000,E1 185.853} C_DIS
LIN {X 0.054,Y -447.205,Z 369.811,A 0.000,B 0.000,C 90.000,E1 181.949} C_DIS
LIN {X -0.205,Y -443.355,Z 369.786,A 0.000,B 0.000,C 90.000,E1 177.421} C_DIS
LIN {X -0.236,Y -441.489,Z 369.756,A 0.000,B 0.000,C 90.000,E1 172.186} C_DIS
LIN {X 0.167,Y -441.643,Z 369.742,A 0.000,B 0.000,C 90.000,E1 169.511} C_DIS
LIN {X 0.100,Y -443.266,Z 369.720,A 0.000,B 0.000,C 90.000,E1 165.589} C_DIS
LIN {X -0.203,Y -445.925,Z 369.702,A 0.000,B 0.000,C 90.000,E1 162.362} C_DIS
LIN {X -0.140,Y -448.780,Z 369.687,A 0.000,B 0.000,C 90.000,E1 159.752} C_DIS
LIN {X 0.227,Y -452.887,Z 369.671,A 0.000,B 0.000,C 90.000,E1 156.794} C_DIS
LIN {X -0.241,Y -458.337,Z 369.653,A 0.000,B 0.000,C 90.000,E1 153.640} C_DIS
LIN {X 0.205,Y -464.308,Z 369.638,A 0.000,B 0.000,C 90.000,E1 150.717} C_DIS
LIN {X 0.055,Y -468.025,Z 369.629,A 0.000,B 0.000,C 90.000,E1 149.154} C_DIS
LIN {X 0.125,Y -478.560,Z 369.608,A 0.000,B 0.000,C 90.000,E1 145.388} C_DIS
LIN {X 0.019,Y -488.707,Z 369.591,A 0.000,B 0.000,C 90.000,E1 142.316} C_DIS
LIN {X -0.088,Y -493.894,Z 369.582,A 0.000,B 0.000,C 90.000,E1 140.803} C_DIS
LIN {X -0.036,Y -497.925,Z 369.576,A 0.000,B 0.000,C 90.000,E1 139.585} C_DIS
LIN {X -0.045,Y -502.818,Z 369.567,A 0.000,B 0.000,C 90.000,E1 138.081} C_DIS
LIN {X 0.260,Y -505.590,Z 369.562,A 0.000,B 0.000,C 90.000,E1 137.148} C_DIS
LIN {X 0.116,Y -509.102,Z 369.556,A 0.000,B 0.000,C 90.000,E1 135.972} C_DIS
LIN {X -0.093,Y -512.990,Z 369.547,A 0.000,B 0.000,C 90.000,E1 134.514} C_DIS
LIN {X -0.042,Y -514.994,Z 369.542,A 0.000,B 0.000,C 90.000,E1 133.623} C_DIS
LIN {X -0.054,Y -517.157,Z 369.536,A 0.000,B 0.000,C 90.000,E1 132.447} C_DIS
LIN {X 0.143,Y -518.148,Z 369.533,A 0.000,B 0.000,C 90.000,E1 131.838} C_DIS
LIN {X -0.105,Y -519.280,Z 369.528,A 0.000,B 0.000,C 90.000,E1 130.987} C_DIS
LIN {X -0.007,Y -520.246,Z 369.521,A 0.000,B 0.000,C 90.000,E1 129.806} C_DIS
LIN {X -0.061,Y -520.412,Z 369.520,A 0.000,B 0.000,C 90.000,E1 129.519} C_DIS
LIN {X 0.111,Y -520.511,Z 369.515,A 0.000,B 0.000,C 90.000,E1 128.624} C_DIS
LIN {X 0.010,Y -520.318,Z 369.511,A 0.000,B 0.000,C 90.000,E1 128.051} C_DIS
LIN {X 0.174,Y -519.756,Z 369.507,A 0.000,B 0.000,C 90.000,E1 127.156} C_DIS
LIN {X -0.043,Y -518.597,Z 369.500,A 0.000,B 0.000,C 90.000,E1 126.011} C_DIS
LIN {X 0.204,Y -517.448,Z 369.495,A 0.000,B 0.000,C 90.000,E1 125.105} C_DIS
LIN {X 0.013,Y -516.064,Z 369.490,A 0.000,B 0.000,C 90.000,E1 124.246} C_DIS
LIN {X -0.058,Y -514.462,Z 369.485,A 0.000,B 0.000,C 90.000,E1 123.372} C_DIS
LIN {X -0.221,Y -512.034,Z 369.479,A 0.000,B 0.000,C 90.000,E1 122.212} C_DIS
LIN {X 0.035,Y -510.633,Z 369.476,A 0.000,B 0.000,C 90.000,E1 121.592} C_DIS
LIN {X -0.128,Y -506.658,Z 369.467,A 0.000,B 0.000,C 90.000,E1 120.129} C_DIS
LIN {X -0.175,Y -504.968,Z 369.464,A 0.000,B 0.000,C 90.000,E1 119.539} C_DIS
LIN {X 0.074,Y -502.182,Z 369.459,A 0.000,B 0.000,C 90.000,E1 118.615} C_DIS
LIN {X -0.006,Y -500.187,Z 369.456,A 0.000,B 0.000,C 90.000,E1 118.025} C_DIS
LIN {X 0.002,Y -495.977,Z 369.449,A 0.000,B 0.000,C 90.000,E1 116.821} C_DIS
LIN {X -0.082,Y -492.575,Z 369.444,A 0.000,B 0.000,C 90.000,E1 115.924} C_DIS
LIN {X 0.030,Y -488.332,Z 369.438,A 0.000,B 0.000,C 90.000,E1 114.847} C_DIS
LIN {X 0.084,Y -482.459,Z 369.430,A 0.000,B 0.000,C 90.000,E1 113.462} C_DIS
LIN {X 0.041,Y -477.563,Z 369.424,A 0.000,B 0.000,C 90.000,E1 112.386} C_DIS
LIN {X 0.188,Y -472.460,Z 369.418,A 0.000,B 0.000,C 90.000,E1 111.280} C_DIS
LIN {X 0.048,Y -465.685,Z 369.411,A 0.000,B 0.000,C 90.000,E1 109.885} C_DIS
LIN {X 0.011,Y -459.537,Z 369.403,A 0.000,B 0.000,C 90.000,E1 108.598} C_DIS
LIN {X -0.028,Y -459.513,Z 369.403,A 0.000,B 0.000,C 90.000,E1 108.598} C_DIS
LIN {X 0.154,Y -467.594,Z 369.383,A 0.000,B 0.000,C 90.000,E1 104.954} C_DIS
LIN {X -0.113,Y -468.592,Z 369.380,A 0.000,B 0.000,C 90.000,E1 104.356} C_DIS
LIN {X 0.113,Y -475.822,Z 369.357,A 0.000,B 0.000,C 90.000,E1 100.254} C_DIS
LIN {X -0.049,Y -476.314,Z 369.355,A 0.000,B 0.000,C 90.000,E1 99.962} C_DIS
LIN {X -0.102,Y -481.805,Z 369.331,A 0.000,B 0.000,C 90.000,E1 95.625} C_DIS
LIN {X 0.226,Y -482.175,Z 369.330,A 0.000,B 0.000,C 90.000,E1 95.277} C_DIS
LIN {X 0.160,Y -485.318,Z 369.306,A 0.000,B 0.000,C 90.000,E1 90.974} C_DIS
LIN {X -0.016,Y -485.536,Z 369.304,A 0.000,B 0.000,C 90.000,E1 90.688} C_DIS
LIN {X 0.191,Y -486.324,Z 369.282,A 0.000,B 0.000,C 90.000,E1 86.674} C_DIS
LIN {X -0.159,Y -486.298,Z 369.278,A 0.000,B 0.000,C 90.000,E1 86.102} C_DIS
LIN {X 0.045,Y -484.695,Z 369.254,A 0.000,B 0.000,C 90.000,E1 81.781} C_DIS
LIN {X -0.086,Y -484.588,Z 369.253,A 0.000,B 0.000,C 90.000,E1 81.489} C_DIS
LIN {X -0.206,Y -480.524,Z 369.227,A 0.000,B 0.000,C 90.000,E1 76.881} C_DIS
LIN {X 0.035,Y -475.218,Z 369.206,A 0.000,B 0.000,C 90.000,E1 73.087} C_DIS
LIN {X -0.005,Y -475.249,Z 369.206,A 0.000,B 0.000,C 90.000,E1 73.087} C_DIS
LIN {X -0.220,Y -484.188,Z 369.199,A 0.000,B 0.000,C 90.000,E1 71.764} C_DIS
LIN {X 0.132,Y -491.927,Z 369.192,A 0.000,B 0.000,C 90.000,E1 70.496} C_DIS
LIN {X 0.254,Y -497.310,Z 369.187,A 0.000,B 0.000,C 90.000,E1 69.571} C_DIS
LIN {X -0.257,Y -500.673,Z 369.183,A 0.000,B 0.000,C 90.000,E1 69.028} C_DIS
LIN {X -0.100,Y -503.608,Z 369.180,A 0.000,B 0.000,C 90.000,E1 68.411} C_DIS
LIN {X -0.020,Y -505.008,Z 369.178,A 0.000,B 0.000,C 90.000,E1 68.103} C_DIS
LIN {X -0.212,Y -505.835,Z 369.178,A 0.000,B 0.000,C 90.000,E1 67.975} C_DIS
LIN {X 0.158,Y -507.748,Z 369.175,A 0.000,B 0.000,C 90.000,E1 67.486} C_DIS
LIN {X -0.214,Y -509.199,Z 369.173,A 0.000,B 0.000,C 90.000,E1 67.230} C_DIS
LIN {X -0.006,Y -511.833,Z 369.170,A 0.000,B 0.000,C 90.000,E1 66.613} C_DIS
LIN {X -0.306,Y -515.900,Z 369.164,A 0.000,B 0.000,C 90.000,E1 65.613} C_DIS
LIN {X 0.033,Y -517.051,Z 369.163,A 0.000,B 0.000,C 90.000,E1 65.281} C_DIS
LIN {X -0.041,Y -519.981,Z 369.158,A 0.000,B 0.000,C 90.000,E1 64.409} C_DIS
LIN {X 0.141,Y -522.751,Z 369.153,A 0.000,B 0.000,C 90.000,E1 63.512} C_DIS
LIN {X -0.273,Y -526.962,Z 369.145,A 0.000,B 0.000,C 90.000,E1 62.103} C_DIS
LIN {X -0.110,Y -531.026,Z 369.137,A 0.000,B 0.000,C 90.000,E1 60.639} C_DIS
LIN {X 0.162,Y -534.211,Z 369.130,A 0.000,B 0.000,C 90.000,E1 59.459} C_DIS
LIN {X 0.013,Y -537.997,Z 369.123,A 0.000,B 0.000,C 90.000,E1 58.043} C_DIS
LIN {X 0.195,Y -540.129,Z 369.118,A 0.000,B 0.000,C 90.000,E1 57.168} C_DIS
LIN {X 0.138,Y -543.588,Z 369.110,A 0.000,B 0.000,C 90.000,E1 55.754} C_DIS
LIN {X 0.230,Y -545.467,Z 369.105,A 0.000,B 0.000,C 90.000,E1 54.895} C_DIS
LIN {X 0.028,Y -547.159,Z 369.100,A 0.000,B 0.000,C 90.000,E1 54.069} C_DIS
LIN {X 0.163,Y -548.625,Z 369.096,A 0.000,B 0.000,C 90.000,E1 53.210} C_DIS
LIN {X -0.067,Y -550.274,Z 369.090,A 0.000,B 0.000,C 90.000,E1 52.110} C_DIS
LIN {X -0.011,Y -550.595,Z 369.088,A 0.000,B 0.000,C 90.000,E1 51.823} C_DIS
LIN {X -0.211,Y -551.481,Z 369.082,A 0.000,B 0.000,C 90.000,E1 50.723} C_DIS
LIN {X -0.095,Y -551.664,Z 369.079,A 0.000,B 0.000,C 90.000,E1 50.150} C_DIS
LIN {X 0.317,Y -551.615,Z 369.077,A 0.000,B 0.000,C 90.000,E1 49.828} C_DIS
LIN {X 0.012,Y -551.821,Z 369.074,A 0.000,B 0.000,C 90.000,E1 49.299} C_DIS
LIN {X 0.127,Y -551.641,Z 369.069,A 0.000,B 0.000,C 90.000,E1 48.447} C_DIS
LIN {X 0.291,Y -550.951,Z 369.063,A 0.000,B 0.000,C 90.000,E1 47.310} C_DIS
LIN {X 0.034,Y -549.799,Z 369.057,A 0.000,B 0.000,C 90.000,E1 46.215} C_DIS
LIN {X 0.188,Y -547.552,Z 369.047,A 0.000,B 0.000,C 90.000,E1 44.514} C_DIS
LIN {X -0.086,Y -545.257,Z 369.038,A 0.000,B 0.000,C 90.000,E1 42.852} C_DIS
LIN {X 0.013,Y -542.561,Z 369.027,A 0.000,B 0.000,C 90.000,E1 40.862} C_DIS
LIN {X -0.327,Y -540.302,Z 369.018,A 0.000,B 0.000,C 90.000,E1 39.197} C_DIS
LIN {X 0.113,Y -538.035,Z 369.008,A 0.000,B 0.000,C 90.000,E1 37.443} C_DIS
LIN {X 0.168,Y -536.192,Z 369.000,A 0.000,B 0.000,C 90.000,E1 36.011} C_DIS
LIN {X -0.128,Y -533.913,Z 368.991,A 0.000,B 0.000,C 90.000,E1 34.326} C_DIS
LIN {X -0.039,Y -531.722,Z 368.981,A 0.000,B 0.000,C 90.000,E1 32.594} C_DIS
LIN {X -0.145,Y -529.233,Z 368.970,A 0.000,B 0.000,C 90.000,E1 30.590} C_DIS
LIN {X -0.111,Y -526.927,Z 368.959,A 0.000,B 0.000,C 90.000,E1 28.565} C_DIS
LIN {X 0.177,Y -524.056,Z 368.944,A 0.000,B 0.000,C 90.000,E1 25.924} C_DIS
LIN {X -0.074,Y -522.273,Z 368.934,A 0.000,B 0.000,C 90.000,E1 24.207} C_DIS
LIN {X -0.258,Y -520.895,Z 368.926,A 0.000,B 0.000,C 90.000,E1 22.770} C_DIS
LIN {X 0.196,Y -520.052,Z 368.922,A 0.000,B 0.000,C 90.000,E1 21.844} C_DIS
LIN {X -0.080,Y -518.746,Z 368.912,A 0.000,B 0.000,C 90.000,E1 20.120} C_DIS
LIN {X 0.156,Y -517.026,Z 368.897,A 0.000,B 0.000,C 90.000,E1 17.457} C_DIS
LIN {X -0.065,Y -516.088,Z 368.886,A 0.000,B 0.000,C 90.000,E1 15.426} C_DIS
LIN {X -0.003,Y -515.285,Z 368.869,A 0.000,B 0.000,C 90.000,E1 12.479} C_DIS
LIN {X -0.162,Y -515.180,Z 368.855,A 0.000,B 0.000,C 90.000,E1 9.849} C_DIS
LIN {X 0.010,Y -515.675,Z 368.840,A 0.000,B 0.000,C 90.000,E1 7.182} C_DIS
LIN {X 0.098,Y -516.672,Z 368.827,A 0.000,B 0.000,C 90.000,E1 4.821} C_DIS
LIN {X 0.176,Y -518.277,Z 368.814,A 0.000,B 0.000,C 90.000,E1 2.465} C_DIS
LIN {X 0.097,Y -521.585,Z 368.796,A 0.000,B 0.000,C 90.000,E1 359.198} C_DIS
LIN {X -0.164,Y -523.920,Z 368.786,A 0.000,B 0.000,C 90.000,E1 357.478} C_DIS
LIN {X 0.122,Y -528.515,Z 368.770,A 0.000,B 0.000,C 90.000,E1 354.546} C_DIS
LIN {X 0.130,Y -533.320,Z 368.755,A 0.000,B 0.000,C 90.000,E1 351.951} C_DIS
LIN {X -0.024,Y -539.547,Z 368.740,A 0.000,B 0.000,C 90.000,E1 349.106} C_DIS
LIN {X -0.020,Y -544.607,Z 368.728,A 0.000,B 0.000,C 90.000,E1 347.117} C_DIS
LIN {X 0.033,Y -548.549,Z 368.721,A 0.000,B 0.000,C 90.000,E1 345.700} C_DIS
LIN {X -0.117,Y -553.437,Z 368.711,A 0.000,B 0.000,C 90.000,E1 344.031} C_DIS
LIN {X -0.035,Y -556.827,Z 368.705,A 0.000,B 0.000,C 90.000,E1 342.906} C_DIS
LIN {X -0.073,Y -562.720,Z 368.694,A 0.000,B 0.000,C 90.000,E1 340.967} C_DIS
LIN {X -0.099,Y -567.853,Z 368.685,A 0.000,B 0.000,C 90.000,E1 339.316} C_DIS
LIN {X -0.023,Y -572.898,Z 368.676,A 0.000,B 0.000,C 90.000,E1 337.667} C_DIS
LIN {X -0.010,Y -577.140,Z 368.668,A 0.000,B 0.000,C 90.000,E1 336.305} C_DIS
LIN {X 0.170,Y -582.265,Z 368.659,A 0.000,B 0.000,C 90.000,E1 334.665} C_DIS
LIN {X -0.146,Y -590.137,Z 368.646,A 0.000,B 0.000,C 90.000,E1 332.281} C_DIS
LIN {X 0.045,Y -595.583,Z 368.637,A 0.000,B 0.000,C 90.000,E1 330.667} C_DIS
LIN {X 0.033,Y -601.948,Z 368.627,A 0.000,B 0.000,C 90.000,E1 328.820} C_DIS
LIN {X -0.223,Y -606.415,Z 368.620,A 0.000,B 0.000,C 90.000,E1 327.533} C_DIS
LIN {X -0.123,Y -614.627,Z 368.607,A 0.000,B 0.000,C 90.000,E1 325.182} C_DIS
LIN {X -0.010,Y -620.269,Z 368.598,A 0.000,B 0.000,C 90.000,E1 323.623} C_DIS
LIN {X -0.120,Y -625.067,Z 368.591,A 0.000,B 0.000,C 90.000,E1 322.351} C_DIS
LIN {X -0.040,Y -631.684,Z 368.581,A 0.000,B 0.000,C 90.000,E1 320.561} C_DIS
LIN {X 0.309,Y -637.485,Z 368.573,A 0.000,B 0.000,C 90.000,E1 319.013} C_DIS
LIN {X -0.025,Y -641.133,Z 368.567,A 0.000,B 0.000,C 90.000,E1 318.038} C_DIS
LIN {X -0.290,Y -650.043,Z 368.553,A 0.000,B 0.000,C 90.000,E1 315.567} C_DIS
LIN {X 0.305,Y -656.408,Z 368.543,A 0.000,B 0.000,C 90.000,E1 313.785} C_DIS
LIN {X -0.246,Y -659.056,Z 368.539,A 0.000,B 0.000,C 90.000,E1 313.095} C_DIS
LIN {X 0.109,Y -664.302,Z 368.531,A 0.000,B 0.000,C 90.000,E1 311.595} C_DIS
LIN {X 0.119,Y -668.530,Z 368.524,A 0.000,B 0.000,C 90.000,E1 310.378} C_DIS
LIN {X 0.288,Y -673.316,Z 368.516,A 0.000,B 0.000,C 90.000,E1 308.910} C_DIS
LIN {X 0.003,Y -676.522,Z 368.511,A 0.000,B 0.000,C 90.000,E1 307.971} C_DIS
LIN {X 0.157,Y -678.765,Z 368.507,A 0.000,B 0.000,C 90.000,E1 307.237} C_DIS
LIN {X -0.063,Y -681.535,Z 368.502,A 0.000,B 0.000,C 90.000,E1 306.297} C_DIS
LIN {X -0.080,Y -684.757,Z 368.495,A 0.000,B 0.000,C 90.000,E1 305.105} C_DIS
LIN {X -0.257,Y -686.566,Z 368.491,A 0.000,B 0.000,C 90.000,E1 304.405} C_DIS
LIN {X 0.166,Y -688.662,Z 368.486,A 0.000,B 0.000,C 90.000,E1 303.420} C_DIS
LIN {X -0.271,Y -691.636,Z 368.477,A 0.000,B 0.000,C 90.000,E1 301.799} C_DIS
LIN {X -0.403,Y -692.407,Z 368.474,A 0.000,B 0.000,C 90.000,E1 301.337} C_DIS
LIN {X 0.305,Y -693.374,Z 368.469,A 0.000,B 0.000,C 90.000,E1 300.335} C_DIS
LIN {X 0.188,Y -693.719,Z 368.466,A 0.000,B 0.000,C 90.000,E1 299.873} C_DIS
LIN {X 0.075,Y -693.941,Z 368.463,A 0.000,B 0.000,C 90.000,E1 299.411} C_DIS
LIN {X -0.037,Y -693.941,Z 368.461,A 0.000,B 0.000,C 90.000,E1 298.949} C_DIS
LIN {X 0.211,Y -693.809,Z 368.460,A 0.000,B 0.000,C 90.000,E1 298.693} C_DIS
LIN {X -0.151,Y -693.838,Z 368.458,A 0.000,B 0.000,C 90.000,E1 298.487} C_DIS
LIN {X -0.266,Y -693.698,Z 368.456,A 0.000,B 0.000,C 90.000,E1 298.025} C_DIS
LIN {X 0.229,Y -693.134,Z 368.453,A 0.000,B 0.000,C 90.000,E1 297.513} C_DIS
LIN {X 0.105,Y -692.838,Z 368.450,A 0.000,B 0.000,C 90.000,E1 297.052} C_DIS
LIN {X 0.154,Y -691.675,Z 368.445,A 0.000,B 0.000,C 90.000,E1 296.104} C_DIS
LIN {X 0.196,Y -690.327,Z 368.440,A 0.000,B 0.000,C 90.000,E1 295.155} C_DIS
LIN {X -0.011,Y -689.117,Z 368.436,A 0.000,B 0.000,C 90.000,E1 294.463} C_DIS
LIN {X 0.218,Y -686.705,Z 368.429,A 0.000,B 0.000,C 90.000,E1 293.259} C_DIS
LIN {X -0.082,Y -684.647,Z 368.424,A 0.000,B 0.000,C 90.000,E1 292.333} C_DIS
LIN {X -0.255,Y -681.220,Z 368.416,A 0.000,B 0.000,C 90.000,E1 290.918} C_DIS
LIN {X 0.252,Y -676.700,Z 368.406,A 0.000,B 0.000,C 90.000,E1 288.960} C_DIS
LIN {X 0.264,Y -672.740,Z 368.396,A 0.000,B 0.000,C 90.000,E1 287.275} C_DIS
LIN {X 0.064,Y -669.414,Z 368.388,A 0.000,B 0.000,C 90.000,E1 285.843} C_DIS
LIN {X 0.201,Y -664.822,Z 368.376,A 0.000,B 0.000,C 90.000,E1 283.647} C_DIS
LIN {X -0.203,Y -660.454,Z 368.362,A 0.000,B 0.000,C 90.000,E1 281.243} C_DIS
LIN {X -0.330,Y -657.006,Z 368.349,A 0.000,B 0.000,C 90.000,E1 278.803} C_DIS
LIN {X 0.286,Y -654.048,Z 368.332,A 0.000,B 0.000,C 90.000,E1 275.796} C_DIS
LIN {X -0.061,Y -652.452,Z 368.316,A 0.000,B 0.000,C 90.000,E1 272.865} C_DIS
LIN {X 0.307,Y -651.876,Z 368.301,A 0.000,B 0.000,C 90.000,E1 270.115} C_DIS
LIN {X -0.187,Y -652.427,Z 368.284,A 0.000,B 0.000,C 90.000,E1 267.192} C_DIS
LIN {X -0.260,Y -653.132,Z 368.275,A 0.000,B 0.000,C 90.000,E1 265.469} C_DIS
LIN {X -0.260,Y -653.838,Z 368.265,A 0.000,B 0.000,C 90.000,E1 263.742} C_DIS
LIN {X -0.166,Y -654.407,Z 368.256,A 0.000,B 0.000,C 90.000,E1 262.008} C_DIS
LIN {X -0.001,Y -654.562,Z 368.251,A 0.000,B 0.000,C 90.000,E1 261.254} C_DIS
LIN {X 0.290,Y -654.474,Z 368.249,A 0.000,B 0.000,C 90.000,E1 260.735} C_DIS
LIN {X -0.165,Y -653.545,Z 368.239,A 0.000,B 0.000,C 90.000,E1 259.050} C_DIS
LIN {X 0.230,Y -653.316,Z 368.236,A 0.000,B 0.000,C 90.000,E1 258.522} C_DIS
LIN {X 0.109,Y -653.109,Z 368.235,A 0.000,B 0.000,C 90.000,E1 258.285} C_DIS
LIN {X -0.013,Y -653.074,Z 368.234,A 0.000,B 0.000,C 90.000,E1 258.049} C_DIS
LIN {X -0.130,Y -652.199,Z 368.227,A 0.000,B 0.000,C 90.000,E1 256.825} C_DIS
LIN {X 0.255,Y -651.755,Z 368.224,A 0.000,B 0.000,C 90.000,E1 256.297} C_DIS
LIN {X -0.088,Y -650.590,Z 368.219,A 0.000,B 0.000,C 90.000,E1 255.338} C_DIS
LIN {X 0.154,Y -649.399,Z 368.214,A 0.000,B 0.000,C 90.000,E1 254.574} C_DIS
LIN {X -0.248,Y -647.975,Z 368.210,A 0.000,B 0.000,C 90.000,E1 253.866} C_DIS
LIN {X 0.137,Y -646.287,Z 368.206,A 0.000,B 0.000,C 90.000,E1 253.087} C_DIS
LIN {X 0.037,Y -645.075,Z 368.203,A 0.000,B 0.000,C 90.000,E1 252.598} C_DIS
LIN {X -0.217,Y -643.014,Z 368.199,A 0.000,B 0.000,C 90.000,E1 251.873} C_DIS
LIN {X 0.118,Y -640.726,Z 368.195,A 0.000,B 0.000,C 90.000,E1 251.094} C_DIS
LIN {X -0.008,Y -639.102,Z 368.192,A 0.000,B 0.000,C 90.000,E1 250.604} C_DIS
LIN {X 0.121,Y -634.485,Z 368.185,A 0.000,B 0.000,C 90.000,E1 249.337} C_DIS
LIN {X 0.009,Y -630.710,Z 368.180,A 0.000,B 0.000,C 90.000,E1 248.337} C_DIS
LIN {X 0.210,Y -625.770,Z 368.173,A 0.000,B 0.000,C 90.000,E1 247.050} C_DIS
LIN {X -0.009,Y -620.505,Z 368.166,A 0.000,B 0.000,C 90.000,E1 245.793} C_DIS
LIN {X -0.312,Y -615.163,Z 368.158,A 0.000,B 0.000,C 90.000,E1 244.537} C_DIS
LIN {X 0.107,Y -609.767,Z 368.151,A 0.000,B 0.000,C 90.000,E1 243.204} C_DIS
LIN {X 0.109,Y -603.387,Z 368.143,A 0.000,B 0.000,C 90.000,E1 241.641} C_DIS
LIN {X -0.016,Y -597.002,Z 368.134,A 0.000,B 0.000,C 90.000,E1 240.078} C_DIS
LIN {X 0.100,Y -588.731,Z 368.122,A 0.000,B 0.000,C 90.000,E1 237.946} C_DIS
LIN {X 0.127,Y -581.009,Z 368.110,A 0.000,B 0.000,C 90.000,E1 235.801} C_DIS
LIN {X 0.284,Y -573.744,Z 368.098,A 0.000,B 0.000,C 90.000,E1 233.623} C_DIS
LIN {X 0.052,Y -570.125,Z 368.092,A 0.000,B 0.000,C 90.000,E1 232.557} C_DIS
LIN {X 0.235,Y -565.346,Z 368.084,A 0.000,B 0.000,C 90.000,E1 231.170} C_DIS
LIN {X -0.259,Y -557.710,Z 368.072,A 0.000,B 0.000,C 90.000,E1 229.013} C_DIS
LIN {X 0.068,Y -552.244,Z 368.063,A 0.000,B 0.000,C 90.000,E1 227.310} C_DIS
LIN {X 0.240,Y -547.722,Z 368.055,A 0.000,B 0.000,C 90.000,E1 225.891} C_DIS
LIN {X -0.061,Y -543.200,Z 368.047,A 0.000,B 0.000,C 90.000,E1 224.514} C_DIS
LIN {X -0.073,Y -537.799,Z 368.038,A 0.000,B 0.000,C 90.000,E1 222.813} C_DIS
LIN {X -0.127,Y -533.463,Z 368.030,A 0.000,B 0.000,C 90.000,E1 221.391} C_DIS
LIN {X 0.030,Y -526.577,Z 368.017,A 0.000,B 0.000,C 90.000,E1 219.072} C_DIS
LIN {X 0.112,Y -520.788,Z 368.006,A 0.000,B 0.000,C 90.000,E1 217.030} C_DIS
LIN {X -0.209,Y -516.056,Z 367.996,A 0.000,B 0.000,C 90.000,E1 215.311} C_DIS
LIN {X 0.086,Y -509.330,Z 367.981,A 0.000,B 0.000,C 90.000,E1 212.625} C_DIS
LIN {X 0.114,Y -504.445,Z 367.970,A 0.000,B 0.000,C 90.000,E1 210.541} C_DIS
LIN {X 0.141,Y -500.380,Z 367.960,A 0.000,B 0.000,C 90.000,E1 208.743} C_DIS
LIN {X -0.133,Y -495.679,Z 367.948,A 0.000,B 0.000,C 90.000,E1 206.668} C_DIS
LIN {X -0.145,Y -492.259,Z 367.940,A 0.000,B 0.000,C 90.000,E1 205.155} C_DIS
LIN {X -0.216,Y -488.792,Z 367.931,A 0.000,B 0.000,C 90.000,E1 203.643} C_DIS
LIN {X 0.103,Y -484.458,Z 367.921,A 0.000,B 0.000,C 90.000,E1 201.770} C_DIS
LIN {X -0.045,Y -479.407,Z 367.909,A 0.000,B 0.000,C 90.000,E1 199.631} C_DIS
LIN {X -0.236,Y -473.277,Z 367.894,A 0.000,B 0.000,C 90.000,E1 196.858} C_DIS
LIN {X -0.074,Y -468.789,Z 367.881,A 0.000,B 0.000,C 90.000,E1 194.647} C_DIS
LIN {X -0.021,Y -463.967,Z 367.867,A 0.000,B 0.000,C 90.000,E1 192.119} C_DIS
LIN {X -0.085,Y -459.989,Z 367.855,A 0.000,B 0.000,C 90.000,E1 189.905} C_DIS
LIN {X 0.190,Y -457.270,Z 367.846,A 0.000,B 0.000,C 90.000,E1 188.276} C_DIS
LIN {X -0.037,Y -453.285,Z 367.832,A 0.000,B 0.000,C 90.000,E1 185.739} C_DIS
LIN {X 0.189,Y -448.317,Z 367.810,A 0.000,B 0.000,C 90.000,E1 181.835} C_DIS
LIN {X -0.146,Y -444.648,Z 367.787,A 0.000,B 0.000,C 90.000,E1 177.650} C_DIS
LIN {X 0.205,Y -443.152,Z 367.771,A 0.000,B 0.000,C 90.000,E1 174.666} C_DIS
LIN {X -0.202,Y -442.628,Z 367.749,A 0.000,B 0.000,C 90.000,E1 170.792} C_DIS
LIN {X -0.161,Y -444.212,Z 367.721,A 0.000,B 0.000,C 90.000,E1 165.880} C_DIS
LIN {X 0.145,Y -446.449,Z 367.705,A 0.000,B 0.000,C 90.000,E1 162.906} C_DIS
LIN {X -0.176,Y -449.932,Z 367.687,A 0.000,B 0.000,C 90.000,E1 159.699} C_DIS
LIN {X -0.194,Y -454.003,Z 367.671,A 0.000,B 0.000,C 90.000,E1 156.794} C_DIS
LIN {X -0.104,Y -460.067,Z 367.651,A 0.000,B 0.000,C 90.000,E1 153.256} C_DIS
LIN {X -0.144,Y -465.463,Z 367.637,A 0.000,B 0.000,C 90.000,E1 150.717} C_DIS
LIN {X 0.097,Y -475.100,Z 367.616,A 0.000,B 0.000,C 90.000,E1 146.914} C_DIS
LIN {X 0.139,Y -483.666,Z 367.601,A 0.000,B 0.000,C 90.000,E1 144.116} C_DIS
LIN {X 0.003,Y -490.931,Z 367.589,A 0.000,B 0.000,C 90.000,E1 141.984} C_DIS
LIN {X 0.241,Y -496.102,Z 367.580,A 0.000,B 0.000,C 90.000,E1 140.436} C_DIS
LIN {X 0.196,Y -501.024,Z 367.572,A 0.000,B 0.000,C 90.000,E1 138.933} C_DIS
LIN {X -0.016,Y -504.855,Z 367.565,A 0.000,B 0.000,C 90.000,E1 137.757} C_DIS
LIN {X 0.200,Y -508.401,Z 367.559,A 0.000,B 0.000,C 90.000,E1 136.539} C_DIS
LIN {X 0.201,Y -510.852,Z 367.554,A 0.000,B 0.000,C 90.000,E1 135.648} C_DIS
LIN {X -0.237,Y -513.895,Z 367.547,A 0.000,B 0.000,C 90.000,E1 134.514} C_DIS
LIN {X -0.175,Y -515.810,Z 367.542,A 0.000,B 0.000,C 90.000,E1 133.623} C_DIS
LIN {X 0.282,Y -517.429,Z 367.537,A 0.000,B 0.000,C 90.000,E1 132.690} C_DIS
LIN {X 0.027,Y -518.842,Z 367.533,A 0.000,B 0.000,C 90.000,E1 131.838} C_DIS
LIN {X -0.215,Y -519.911,Z 367.528,A 0.000,B 0.000,C 90.000,E1 130.987} C_DIS
LIN {X -0.053,Y -520.641,Z 367.523,A 0.000,B 0.000,C 90.000,E1 130.092} C_DIS
LIN {X 0.173,Y -520.966,Z 367.520,A 0.000,B 0.000,C 90.000,E1 129.483} C_DIS
LIN {X 0.019,Y -520.951,Z 367.515,A 0.000,B 0.000,C 90.000,E1 128.624} C_DIS
LIN {X 0.192,Y -520.513,Z 367.510,A 0.000,B 0.000,C 90.000,E1 127.729} C_DIS
LIN {X 0.039,Y -519.748,Z 367.505,A 0.000,B 0.000,C 90.000,E1 126.870} C_DIS
LIN {X -0.179,Y -518.407,Z 367.498,A 0.000,B 0.000,C 90.000,E1 125.724} C_DIS
LIN {X 0.066,Y -517.183,Z 367.494,A 0.000,B 0.000,C 90.000,E1 124.818} C_DIS
LIN {X -0.060,Y -515.205,Z 367.487,A 0.000,B 0.000,C 90.000,E1 123.658} C_DIS
LIN {X 0.065,Y -512.830,Z 367.480,A 0.000,B 0.000,C 90.000,E1 122.467} C_DIS
LIN {X -0.035,Y -510.863,Z 367.476,A 0.000,B 0.000,C 90.000,E1 121.592} C_DIS
LIN {X -0.083,Y -507.777,Z 367.469,A 0.000,B 0.000,C 90.000,E1 120.413} C_DIS
LIN {X -0.237,Y -505.389,Z 367.464,A 0.000,B 0.000,C 90.000,E1 119.539} C_DIS
LIN {X 0.018,Y -502.678,Z 367.459,A 0.000,B 0.000,C 90.000,E1 118.615} C_DIS
LIN {X -0.059,Y -500.761,Z 367.456,A 0.000,B 0.000,C 90.000,E1 118.025} C_DIS
LIN {X -0.042,Y -496.632,Z 367.449,A 0.000,B 0.000,C 90.000,E1 116.821} C_DIS
LIN {X -0.119,Y -493.291,Z 367.444,A 0.000,B 0.000,C 90.000,E1 115.924} C_DIS
LIN {X -0.234,Y -489.717,Z 367.439,A 0.000,B 0.000,C 90.000,E1 115.027} C_DIS
LIN {X -0.168,Y -485.354,Z 367.433,A 0.000,B 0.000,C 90.000,E1 113.951} C_DIS
LIN {X 0.270,Y -479.439,Z 367.425,A 0.000,B 0.000,C 90.000,E1 112.514} C_DIS
LIN {X -0.029,Y -473.002,Z 367.418,A 0.000,B 0.000,C 90.000,E1 111.153} C_DIS
LIN {X 0.036,Y -465.604,Z 367.409,A 0.000,B 0.000,C 90.000,E1 109.577} C_DIS
LIN {X 0.131,Y -459.953,Z 367.402,A 0.000,B 0.000,C 90.000,E1 108.362} C_DIS
LIN {X 0.091,Y -459.944,Z 367.402,A 0.000,B 0.000,C 90.000,E1 108.362} C_DIS
LIN {X -0.225,Y -467.571,Z 367.383,A 0.000,B 0.000,C 90.000,E1 105.009} C_DIS
LIN {X -0.042,Y -468.579,Z 367.380,A 0.000,B 0.000,C 90.000,E1 104.356} C_DIS
LIN {X 0.185,Y -475.804,Z 367.357,A 0.000,B 0.000,C 90.000,E1 100.254} C_DIS
LIN {X 0.024,Y -476.306,Z 367.355,A 0.000,B 0.000,C 90.000,E1 99.962} C_DIS
LIN {X -0.029,Y -481.791,Z 367.331,A 0.000,B 0.000,C 90.000,E1 95.625} C_DIS
LIN {X -0.182,Y -482.171,Z 367.330,A 0.000,B 0.000,C 90.000,E1 95.334} C_DIS
LIN {X 0.232,Y -485.309,Z 367.306,A 0.000,B 0.000,C 90.000,E1 90.974} C_DIS
LIN {X 0.057,Y -485.537,Z 367.304,A 0.000,B 0.000,C 90.000,E1 90.688} C_DIS
LIN {X -0.222,Y -486.320,Z 367.282,A 0.000,B 0.000,C 90.000,E1 86.731} C_DIS
LIN {X -0.087,Y -486.304,Z 367.278,A 0.000,B 0.000,C 90.000,E1 86.102} C_DIS
LIN {X 0.118,Y -484.696,Z 367.254,A 0.000,B 0.000,C 90.000,E1 81.781} C_DIS
LIN {X -0.013,Y -484.599,Z 367.253,A 0.000,B 0.000,C 90.000,E1 81.489} C_DIS
LIN {X -0.134,Y -480.533,Z 367.227,A 0.000,B 0.000,C 90.000,E1 76.881} C_DIS
LIN {X -0.104,Y -475.404,Z 367.207,A 0.000,B 0.000,C 90.000,E1 73.268} C_DIS
LIN {X -0.144,Y -475.414,Z 367.207,A 0.000,B 0.000,C 90.000,E1 73.268} C_DIS
LIN {X -0.284,Y -484.102,Z 367.200,A 0.000,B 0.000,C 90.000,E1 71.945} C_DIS
LIN {X -0.153,Y -492.547,Z 367.192,A 0.000,B 0.000,C 90.000,E1 70.550} C_DIS
LIN {X 0.181,Y -496.992,Z 367.188,A 0.000,B 0.000,C 90.000,E1 69.752} C_DIS
LIN {X 0.122,Y -500.319,Z 367.184,A 0.000,B 0.000,C 90.000,E1 69.156} C_DIS
LIN {X 0.068,Y -504.000,Z 367.180,A 0.000,B 0.000,C 90.000,E1 68.411} C_DIS
LIN {X -0.232,Y -506.725,Z 367.177,A 0.000,B 0.000,C 90.000,E1 67.847} C_DIS
LIN {X -0.195,Y -512.148,Z 367.170,A 0.000,B 0.000,C 90.000,E1 66.538} C_DIS
LIN {X 0.209,Y -513.801,Z 367.167,A 0.000,B 0.000,C 90.000,E1 66.049} C_DIS
LIN {X 0.032,Y -514.408,Z 367.166,A 0.000,B 0.000,C 90.000,E1 65.921} C_DIS
LIN {X 0.152,Y -515.378,Z 367.165,A 0.000,B 0.000,C 90.000,E1 65.613} C_DIS
LIN {X -0.194,Y -516.537,Z 367.163,A 0.000,B 0.000,C 90.000,E1 65.357} C_DIS
LIN {X -0.055,Y -519.393,Z 367.158,A 0.000,B 0.000,C 90.000,E1 64.460} C_DIS
LIN {X -0.108,Y -522.140,Z 367.153,A 0.000,B 0.000,C 90.000,E1 63.589} C_DIS
LIN {X 0.170,Y -526.307,Z 367.145,A 0.000,B 0.000,C 90.000,E1 62.103} C_DIS
LIN {X 0.064,Y -530.359,Z 367.137,A 0.000,B 0.000,C 90.000,E1 60.667} C_DIS
LIN {X 0.295,Y -534.330,Z 367.129,A 0.000,B 0.000,C 90.000,E1 59.203} C_DIS
LIN {X 0.144,Y -538.109,Z 367.121,A 0.000,B 0.000,C 90.000,E1 57.788} C_DIS
LIN {X 0.054,Y -541.685,Z 367.113,A 0.000,B 0.000,C 90.000,E1 56.373} C_DIS
LIN {X -0.159,Y -544.398,Z 367.107,A 0.000,B 0.000,C 90.000,E1 55.261} C_DIS
LIN {X -0.017,Y -546.769,Z 367.101,A 0.000,B 0.000,C 90.000,E1 54.116} C_DIS
LIN {X 0.118,Y -548.348,Z 367.096,A 0.000,B 0.000,C 90.000,E1 53.256} C_DIS
LIN {X -0.162,Y -548.725,Z 367.094,A 0.000,B 0.000,C 90.000,E1 53.004} C_DIS
LIN {X -0.064,Y -549.758,Z 367.091,A 0.000,B 0.000,C 90.000,E1 52.431} C_DIS
LIN {X 0.041,Y -550.574,Z 367.088,A 0.000,B 0.000,C 90.000,E1 51.859} C_DIS
LIN {X 0.124,Y -551.388,Z 367.083,A 0.000,B 0.000,C 90.000,E1 51.009} C_DIS
LIN {X -0.125,Y -551.949,Z 367.079,A 0.000,B 0.000,C 90.000,E1 50.194} C_DIS
LIN {X 0.049,Y -552.255,Z 367.074,A 0.000,B 0.000,C 90.000,E1 49.337} C_DIS
LIN {X 0.163,Y -552.168,Z 367.070,A 0.000,B 0.000,C 90.000,E1 48.485} C_DIS
LIN {X -0.129,Y -551.737,Z 367.065,A 0.000,B 0.000,C 90.000,E1 47.676} C_DIS
LIN {X -0.032,Y -551.409,Z 367.062,A 0.000,B 0.000,C 90.000,E1 47.106} C_DIS
LIN {X -0.326,Y -550.608,Z 367.057,A 0.000,B 0.000,C 90.000,E1 46.296} C_DIS
LIN {X 0.208,Y -548.846,Z 367.049,A 0.000,B 0.000,C 90.000,E1 44.838} C_DIS
LIN {X -0.066,Y -547.016,Z 367.041,A 0.000,B 0.000,C 90.000,E1 43.461} C_DIS
LIN {X 0.044,Y -544.681,Z 367.032,A 0.000,B 0.000,C 90.000,E1 41.757} C_DIS
LIN {X -0.228,Y -542.066,Z 367.021,A 0.000,B 0.000,C 90.000,E1 39.806} C_DIS
LIN {X -0.147,Y -539.412,Z 367.010,A 0.000,B 0.000,C 90.000,E1 37.810} C_DIS
LIN {X -0.052,Y -537.160,Z 367.001,A 0.000,B 0.000,C 90.000,E1 36.091} C_DIS
LIN {X -0.324,Y -534.891,Z 366.991,A 0.000,B 0.000,C 90.000,E1 34.405} C_DIS
LIN {X -0.206,Y -532.726,Z 366.981,A 0.000,B 0.000,C 90.000,E1 32.673} C_DIS
LIN {X 0.018,Y -530.571,Z 366.972,A 0.000,B 0.000,C 90.000,E1 30.924} C_DIS
LIN {X -0.074,Y -528.536,Z 366.962,A 0.000,B 0.000,C 90.000,E1 29.205} C_DIS
LIN {X 0.146,Y -527.256,Z 366.956,A 0.000,B 0.000,C 90.000,E1 28.025} C_DIS
LIN {X -0.122,Y -525.073,Z 366.945,A 0.000,B 0.000,C 90.000,E1 26.027} C_DIS
LIN {X 0.112,Y -523.326,Z 366.935,A 0.000,B 0.000,C 90.000,E1 24.259} C_DIS
LIN {X 0.097,Y -521.663,Z 366.925,A 0.000,B 0.000,C 90.000,E1 22.514} C_DIS
LIN {X 0.145,Y -519.797,Z 366.912,A 0.000,B 0.000,C 90.000,E1 20.174} C_DIS
LIN {X -0.218,Y -518.244,Z 366.899,A 0.000,B 0.000,C 90.000,E1 17.873} C_DIS
LIN {X 0.106,Y -517.398,Z 366.889,A 0.000,B 0.000,C 90.000,E1 16.079} C_DIS
LIN {X -0.244,Y -516.626,Z 366.878,A 0.000,B 0.000,C 90.000,E1 14.064} C_DIS
LIN {X -0.244,Y -516.271,Z 366.865,A 0.000,B 0.000,C 90.000,E1 11.715} C_DIS
LIN {X 0.160,Y -516.289,Z 366.854,A 0.000,B 0.000,C 90.000,E1 9.613} C_DIS
LIN {X 0.029,Y -516.333,Z 366.849,A 0.000,B 0.000,C 90.000,E1 8.746} C_DIS
LIN {X -0.114,Y -516.723,Z 366.842,A 0.000,B 0.000,C 90.000,E1 7.587} C_DIS
LIN {X -0.179,Y -518.354,Z 366.823,A 0.000,B 0.000,C 90.000,E1 4.073} C_DIS
LIN {X -0.168,Y -520.721,Z 366.806,A 0.000,B 0.000,C 90.000,E1 1.146} C_DIS
LIN {X -0.089,Y -524.782,Z 366.788,A 0.000,B 0.000,C 90.000,E1 357.764} C_DIS
LIN {X 0.211,Y -528.306,Z 366.775,A 0.000,B 0.000,C 90.000,E1 355.412} C_DIS
LIN {X 0.199,Y -531.835,Z 366.763,A 0.000,B 0.000,C 90.000,E1 353.394} C_DIS
LIN {X -0.252,Y -535.747,Z 366.752,A 0.000,B 0.000,C 90.000,E1 351.432} C_DIS
LIN {X 0.151,Y -540.854,Z 366.740,A 0.000,B 0.000,C 90.000,E1 349.106} C_DIS
LIN {X -0.063,Y -548.290,Z 366.724,A 0.000,B 0.000,C 90.000,E1 346.297} C_DIS
LIN {X 0.149,Y -554.759,Z 366.711,A 0.000,B 0.000,C 90.000,E1 344.031} C_DIS
LIN {X -0.160,Y -558.981,Z 366.704,A 0.000,B 0.000,C 90.000,E1 342.670} C_DIS
LIN {X 0.249,Y -564.056,Z 366.694,A 0.000,B 0.000,C 90.000,E1 340.967} C_DIS
LIN {X -0.086,Y -568.366,Z 366.687,A 0.000,B 0.000,C 90.000,E1 339.625} C_DIS
LIN {X 0.002,Y -573.434,Z 366.678,A 0.000,B 0.000,C 90.000,E1 337.975} C_DIS
LIN {X -0.126,Y -578.569,Z 366.669,A 0.000,B 0.000,C 90.000,E1 336.357} C_DIS
LIN {X 0.090,Y -583.724,Z 366.660,A 0.000,B 0.000,C 90.000,E1 334.717} C_DIS
LIN {X 0.080,Y -591.623,Z 366.646,A 0.000,B 0.000,C 90.000,E1 332.308} C_DIS
LIN {X 0.053,Y -594.349,Z 366.642,A 0.000,B 0.000,C 90.000,E1 331.513} C_DIS
LIN {X -0.115,Y -598.861,Z 366.634,A 0.000,B 0.000,C 90.000,E1 330.205} C_DIS
LIN {X 0.021,Y -604.340,Z 366.626,A 0.000,B 0.000,C 90.000,E1 328.614} C_DIS
LIN {X -0.193,Y -608.833,Z 366.618,A 0.000,B 0.000,C 90.000,E1 327.327} C_DIS
LIN {X 0.034,Y -616.135,Z 366.607,A 0.000,B 0.000,C 90.000,E1 325.229} C_DIS
LIN {X -0.179,Y -621.781,Z 366.598,A 0.000,B 0.000,C 90.000,E1 323.703} C_DIS
LIN {X 0.075,Y -627.522,Z 366.590,A 0.000,B 0.000,C 90.000,E1 322.145} C_DIS
LIN {X 0.093,Y -635.033,Z 366.578,A 0.000,B 0.000,C 90.000,E1 320.114} C_DIS
LIN {X 0.121,Y -639.846,Z 366.572,A 0.000,B 0.000,C 90.000,E1 318.852} C_DIS
LIN {X -0.264,Y -644.283,Z 366.565,A 0.000,B 0.000,C 90.000,E1 317.634} C_DIS
LIN {X -0.372,Y -652.323,Z 366.552,A 0.000,B 0.000,C 90.000,E1 315.405} C_DIS
LIN {X 0.308,Y -657.693,Z 366.544,A 0.000,B 0.000,C 90.000,E1 313.866} C_DIS
LIN {X -0.276,Y -662.016,Z 366.537,A 0.000,B 0.000,C 90.000,E1 312.690} C_DIS
LIN {X 0.151,Y -665.525,Z 366.532,A 0.000,B 0.000,C 90.000,E1 311.676} C_DIS
LIN {X 0.181,Y -669.620,Z 366.525,A 0.000,B 0.000,C 90.000,E1 310.458} C_DIS
LIN {X -0.155,Y -673.613,Z 366.518,A 0.000,B 0.000,C 90.000,E1 309.277} C_DIS
LIN {X 0.104,Y -677.528,Z 366.512,A 0.000,B 0.000,C 90.000,E1 308.051} C_DIS
LIN {X -0.270,Y -679.692,Z 366.508,A 0.000,B 0.000,C 90.000,E1 307.363} C_DIS
LIN {X 0.064,Y -682.356,Z 366.502,A 0.000,B 0.000,C 90.000,E1 306.377} C_DIS
LIN {X -0.116,Y -684.886,Z 366.497,A 0.000,B 0.000,C 90.000,E1 305.438} C_DIS
LIN {X -0.103,Y -687.205,Z 366.492,A 0.000,B 0.000,C 90.000,E1 304.485} C_DIS
LIN {X 0.333,Y -689.207,Z 366.486,A 0.000,B 0.000,C 90.000,E1 303.499} C_DIS
LIN {X 0.271,Y -691.620,Z 366.478,A 0.000,B 0.000,C 90.000,E1 302.084} C_DIS
LIN {X 0.146,Y -692.737,Z 366.474,A 0.000,B 0.000,C 90.000,E1 301.386} C_DIS
LIN {X -0.097,Y -693.705,Z 366.469,A 0.000,B 0.000,C 90.000,E1 300.463} C_DIS
LIN {X -0.213,Y -694.065,Z 366.467,A 0.000,B 0.000,C 90.000,E1 300.001} C_DIS
LIN {X -0.324,Y -694.228,Z 366.464,A 0.000,B 0.000,C 90.000,E1 299.539} C_DIS
LIN {X -0.187,Y -694.134,Z 366.460,A 0.000,B 0.000,C 90.000,E1 298.821} C_DIS
LIN {X -0.050,Y -693.676,Z 366.456,A 0.000,B 0.000,C 90.000,E1 298.103} C_DIS
LIN {X 0.081,Y -692.768,Z 366.452,A 0.000,B 0.000,C 90.000,E1 297.385} C_DIS
LIN {X -0.046,Y -692.365,Z 366.450,A 0.000,B 0.000,C 90.000,E1 296.924} C_DIS
LIN {X -0.147,Y -690.268,Z 366.442,A 0.000,B 0.000,C 90.000,E1 295.515} C_DIS
LIN {X 0.264,Y -689.026,Z 366.438,A 0.000,B 0.000,C 90.000,E1 294.771} C_DIS
LIN {X 0.216,Y -686.596,Z 366.431,A 0.000,B 0.000,C 90.000,E1 293.590} C_DIS
LIN {X 0.187,Y -684.542,Z 366.426,A 0.000,B 0.000,C 90.000,E1 292.642} C_DIS
LIN {X 0.062,Y -681.691,Z 366.419,A 0.000,B 0.000,C 90.000,E1 291.461} C_DIS
LIN {X -0.179,Y -678.207,Z 366.411,A 0.000,B 0.000,C 90.000,E1 290.047} C_DIS
LIN {X -0.237,Y -675.401,Z 366.405,A 0.000,B 0.000,C 90.000,E1 288.852} C_DIS
LIN {X -0.109,Y -670.807,Z 366.394,A 0.000,B 0.000,C 90.000,E1 286.913} C_DIS
LIN {X -0.198,Y -668.592,Z 366.389,A 0.000,B 0.000,C 90.000,E1 285.953} C_DIS
LIN {X -0.255,Y -663.960,Z 366.376,A 0.000,B 0.000,C 90.000,E1 283.772} C_DIS
LIN {X 0.315,Y -658.452,Z 366.359,A 0.000,B 0.000,C 90.000,E1 280.546} C_DIS
LIN {X 0.291,Y -654.452,Z 366.341,A 0.000,B 0.000,C 90.000,E1 277.352} C_DIS
LIN {X 0.283,Y -651.859,Z 366.322,A 0.000,B 0.000,C 90.000,E1 273.898} C_DIS
LIN {X -0.288,Y -651.315,Z 366.314,A 0.000,B 0.000,C 90.000,E1 272.465} C_DIS
LIN {X 0.255,Y -650.874,Z 366.300,A 0.000,B 0.000,C 90.000,E1 269.943} C_DIS
LIN {X -0.069,Y -651.434,Z 366.285,A 0.000,B 0.000,C 90.000,E1 267.249} C_DIS
LIN {X 0.049,Y -652.049,Z 366.276,A 0.000,B 0.000,C 90.000,E1 265.755} C_DIS
LIN {X -0.185,Y -652.882,Z 366.266,A 0.000,B 0.000,C 90.000,E1 263.799} C_DIS
LIN {X -0.336,Y -653.622,Z 366.255,A 0.000,B 0.000,C 90.000,E1 261.837} C_DIS
LIN {X -0.183,Y -653.762,Z 366.250,A 0.000,B 0.000,C 90.000,E1 261.084} C_DIS
LIN {X 0.206,Y -653.658,Z 366.248,A 0.000,B 0.000,C 90.000,E1 260.557} C_DIS
LIN {X -0.131,Y -653.218,Z 366.239,A 0.000,B 0.000,C 90.000,E1 259.106} C_DIS
LIN {X 0.140,Y -652.902,Z 366.235,A 0.000,B 0.000,C 90.000,E1 258.342} C_DIS
LIN {X -0.117,Y -652.916,Z 366.234,A 0.000,B 0.000,C 90.000,E1 258.117} C_DIS
LIN {X -0.096,Y -652.452,Z 366.227,A 0.000,B 0.000,C 90.000,E1 256.881} C_DIS
LIN {X 0.042,Y -651.567,Z 366.222,A 0.000,B 0.000,C 90.000,E1 255.880} C_DIS
LIN {X -0.337,Y -650.715,Z 366.217,A 0.000,B 0.000,C 90.000,E1 255.172} C_DIS
LIN {X 0.074,Y -649.547,Z 366.213,A 0.000,B 0.000,C 90.000,E1 254.393} C_DIS
LIN {X -0.326,Y -648.177,Z 366.209,A 0.000,B 0.000,C 90.000,E1 253.685} C_DIS
LIN {X 0.061,Y -646.569,Z 366.205,A 0.000,B 0.000,C 90.000,E1 252.906} C_DIS
LIN {X -0.034,Y -645.427,Z 366.202,A 0.000,B 0.000,C 90.000,E1 252.417} C_DIS
LIN {X 0.326,Y -643.443,Z 366.198,A 0.000,B 0.000,C 90.000,E1 251.638} C_DIS
LIN {X 0.054,Y -641.205,Z 366.194,A 0.000,B 0.000,C 90.000,E1 250.913} C_DIS
LIN {X -0.069,Y -639.595,Z 366.191,A 0.000,B 0.000,C 90.000,E1 250.423} C_DIS
LIN {X 0.067,Y -635.068,Z 366.184,A 0.000,B 0.000,C 90.000,E1 249.156} C_DIS
LIN {X -0.038,Y -631.326,Z 366.179,A 0.000,B 0.000,C 90.000,E1 248.156} C_DIS
LIN {X 0.170,Y -626.380,Z 366.172,A 0.000,B 0.000,C 90.000,E1 246.869} C_DIS
LIN {X -0.042,Y -621.164,Z 366.165,A 0.000,B 0.000,C 90.000,E1 245.613} C_DIS
LIN {X -0.087,Y -614.794,Z 366.156,A 0.000,B 0.000,C 90.000,E1 244.076} C_DIS
LIN {X 0.247,Y -607.325,Z 366.146,A 0.000,B 0.000,C 90.000,E1 242.231} C_DIS
LIN {X 0.199,Y -600.919,Z 366.137,A 0.000,B 0.000,C 90.000,E1 240.667} C_DIS
LIN {X -0.194,Y -594.605,Z 366.128,A 0.000,B 0.000,C 90.000,E1 239.125} C_DIS
LIN {X 0.053,Y -585.645,Z 366.115,A 0.000,B 0.000,C 90.000,E1 236.707} C_DIS
LIN {X 0.163,Y -577.303,Z 366.102,A 0.000,B 0.000,C 90.000,E1 234.276} C_DIS
LIN {X 0.126,Y -572.822,Z 366.094,A 0.000,B 0.000,C 90.000,E1 232.924} C_DIS
LIN {X 0.093,Y -570.029,Z 366.090,A 0.000,B 0.000,C 90.000,E1 232.110} C_DIS
LIN {X -0.046,Y -564.219,Z 366.080,A 0.000,B 0.000,C 90.000,E1 230.481} C_DIS
LIN {X 0.223,Y -556.711,Z 366.068,A 0.000,B 0.000,C 90.000,E1 228.243} C_DIS
LIN {X 0.041,Y -553.091,Z 366.062,A 0.000,B 0.000,C 90.000,E1 227.148} C_DIS
LIN {X -0.188,Y -549.481,Z 366.056,A 0.000,B 0.000,C 90.000,E1 226.053} C_DIS
LIN {X -0.072,Y -544.953,Z 366.048,A 0.000,B 0.000,C 90.000,E1 224.636} C_DIS
LIN {X -0.029,Y -539.573,Z 366.039,A 0.000,B 0.000,C 90.000,E1 222.933} C_DIS
LIN {X -0.091,Y -534.306,Z 366.029,A 0.000,B 0.000,C 90.000,E1 221.229} C_DIS
LIN {X 0.107,Y -528.261,Z 366.018,A 0.000,B 0.000,C 90.000,E1 219.197} C_DIS
LIN {X 0.261,Y -523.263,Z 366.008,A 0.000,B 0.000,C 90.000,E1 217.443} C_DIS
LIN {X -0.068,Y -517.702,Z 365.997,A 0.000,B 0.000,C 90.000,E1 215.438} C_DIS
LIN {X 0.271,Y -510.905,Z 365.982,A 0.000,B 0.000,C 90.000,E1 212.752} C_DIS
LIN {X -0.102,Y -506.024,Z 365.971,A 0.000,B 0.000,C 90.000,E1 210.718} C_DIS
LIN {X 0.012,Y -501.279,Z 365.959,A 0.000,B 0.000,C 90.000,E1 208.615} C_DIS
LIN {X -0.068,Y -497.273,Z 365.949,A 0.000,B 0.000,C 90.000,E1 206.821} C_DIS
LIN {X 0.172,Y -493.878,Z 365.941,A 0.000,B 0.000,C 90.000,E1 205.283} C_DIS
LIN {X 0.130,Y -490.474,Z 365.932,A 0.000,B 0.000,C 90.000,E1 203.770} C_DIS
LIN {X -0.146,Y -486.165,Z 365.922,A 0.000,B 0.000,C 90.000,E1 201.972} C_DIS
LIN {X -0.070,Y -481.823,Z 365.912,A 0.000,B 0.000,C 90.000,E1 200.120} C_DIS
LIN {X 0.015,Y -476.930,Z 365.900,A 0.000,B 0.000,C 90.000,E1 197.946} C_DIS
LIN {X 0.047,Y -473.641,Z 365.891,A 0.000,B 0.000,C 90.000,E1 196.386} C_DIS
LIN {X 0.064,Y -471.108,Z 365.884,A 0.000,B 0.000,C 90.000,E1 195.134} C_DIS
LIN {X -0.148,Y -466.209,Z 365.870,A 0.000,B 0.000,C 90.000,E1 192.647} C_DIS
LIN {X -0.066,Y -462.168,Z 365.858,A 0.000,B 0.000,C 90.000,E1 190.423} C_DIS
LIN {X 0.176,Y -459.453,Z 365.849,A 0.000,B 0.000,C 90.000,E1 188.803} C_DIS
LIN {X -0.159,Y -454.864,Z 365.833,A 0.000,B 0.000,C 90.000,E1 185.967} C_DIS
LIN {X 0.044,Y -452.123,Z 365.822,A 0.000,B 0.000,C 90.000,E1 184.012} C_DIS
LIN {X -0.130,Y -448.404,Z 365.804,A 0.000,B 0.000,C 90.000,E1 180.802} C_DIS
LIN {X 0.148,Y -445.548,Z 365.785,A 0.000,B 0.000,C 90.000,E1 177.192} C_DIS
LIN {X 0.119,Y -444.184,Z 365.768,A 0.000,B 0.000,C 90.000,E1 174.261} C_DIS
LIN {X 0.202,Y -443.808,Z 365.746,A 0.000,B 0.000,C 90.000,E1 170.330} C_DIS
LIN {X 0.237,Y -445.346,Z 365.721,A 0.000,B 0.000,C 90.000,E1 165.755} C_DIS
LIN {X 0.036,Y -447.563,Z 365.705,A 0.000,B 0.000,C 90.000,E1 162.851} C_DIS
LIN {X 0.213,Y -451.480,Z 365.685,A 0.000,B 0.000,C 90.000,E1 159.263} C_DIS
LIN {X 0.157,Y -456.120,Z 365.667,A 0.000,B 0.000,C 90.000,E1 156.049} C_DIS
LIN {X -0.111,Y -461.225,Z 365.651,A 0.000,B 0.000,C 90.000,E1 153.204} C_DIS
LIN {X 0.022,Y -467.313,Z 365.635,A 0.000,B 0.000,C 90.000,E1 150.333} C_DIS
LIN {X -0.058,Y -477.203,Z 365.614,A 0.000,B 0.000,C 90.000,E1 146.580} C_DIS
LIN {X -0.166,Y -484.893,Z 365.601,A 0.000,B 0.000,C 90.000,E1 144.116} C_DIS
LIN {X 0.028,Y -492.150,Z 365.589,A 0.000,B 0.000,C 90.000,E1 141.949} C_DIS
LIN {X -0.016,Y -497.276,Z 365.580,A 0.000,B 0.000,C 90.000,E1 140.436} C_DIS
LIN {X -0.042,Y -502.163,Z 365.572,A 0.000,B 0.000,C 90.000,E1 138.933} C_DIS
LIN {X 0.254,Y -505.035,Z 365.567,A 0.000,B 0.000,C 90.000,E1 138.000} C_DIS
LIN {X 0.105,Y -508.594,Z 365.560,A 0.000,B 0.000,C 90.000,E1 136.824} C_DIS
LIN {X -0.245,Y -511.081,Z 365.555,A 0.000,B 0.000,C 90.000,E1 135.972} C_DIS
LIN {X 0.045,Y -514.075,Z 365.549,A 0.000,B 0.000,C 90.000,E1 134.757} C_DIS
LIN {X 0.110,Y -516.072,Z 365.544,A 0.000,B 0.000,C 90.000,E1 133.866} C_DIS
LIN {X 0.116,Y -518.144,Z 365.537,A 0.000,B 0.000,C 90.000,E1 132.690} C_DIS
LIN {X -0.132,Y -519.438,Z 365.532,A 0.000,B 0.000,C 90.000,E1 131.838} C_DIS
LIN {X 0.308,Y -520.658,Z 365.526,A 0.000,B 0.000,C 90.000,E1 130.620} C_DIS
LIN {X 0.028,Y -521.257,Z 365.519,A 0.000,B 0.000,C 90.000,E1 129.483} C_DIS
LIN {X -0.122,Y -521.184,Z 365.515,A 0.000,B 0.000,C 90.000,E1 128.624} C_DIS
LIN {X 0.053,Y -520.705,Z 365.510,A 0.000,B 0.000,C 90.000,E1 127.729} C_DIS
LIN {X -0.098,Y -519.910,Z 365.505,A 0.000,B 0.000,C 90.000,E1 126.870} C_DIS
LIN {X 0.108,Y -518.534,Z 365.498,A 0.000,B 0.000,C 90.000,E1 125.678} C_DIS
LIN {X -0.066,Y -517.292,Z 365.493,A 0.000,B 0.000,C 90.000,E1 124.818} C_DIS
LIN {X 0.095,Y -515.311,Z 365.487,A 0.000,B 0.000,C 90.000,E1 123.627} C_DIS
LIN {X 0.019,Y -513.549,Z 365.482,A 0.000,B 0.000,C 90.000,E1 122.752} C_DIS
LIN {X -0.162,Y -510.994,Z 365.475,A 0.000,B 0.000,C 90.000,E1 121.592} C_DIS
LIN {X 0.050,Y -507.935,Z 365.469,A 0.000,B 0.000,C 90.000,E1 120.384} C_DIS
LIN {X 0.082,Y -505.550,Z 365.464,A 0.000,B 0.000,C 90.000,E1 119.489} C_DIS
LIN {X -0.035,Y -501.926,Z 365.457,A 0.000,B 0.000,C 90.000,E1 118.309} C_DIS
LIN {X 0.120,Y -495.956,Z 365.447,A 0.000,B 0.000,C 90.000,E1 116.488} C_DIS
